version 1.4		05. may. 2012
programmer 		ks
tested by		ks

MB_SERVER ermöglicht das Lesen/Schreiben von Daten durch ein Remote-Device mittels Modbus over Ethernet (OpenModbus)

*)
(* read system time *)
tx := DWORD_TO_TIME(T_PLC_MS());

FOR i := 1 TO 10 DO
	IF VMAP[i].TIME_OUT > T#0s THEN
		VMAP[i].TIME_OUT := VMAP[i].TIME_OUT + tx - last_cycle;
	END_IF;
END_FOR;
last_cycle := tx;
ip_error := IP_C.ERROR > DWORD#0;

CASE state OF
00: (* Warten auf Freigabe *)
	IF ENABLE THEN
		state := 10;
		ip_state := BYTE#1; (* Anmelden *)
	END_IF;

10: (* Bei IP_Control anmelden und auf freigabe warten *)
	IF ip_state = BYTE#3 THEN

		(* IP Datenverkehr einrichten *)
		IP_C.C_PORT := WORD#0; (* Port von IP_CONTROL verwenden *)
		IP_C.C_IP := DWORD#0; (* IP von IP_CONTROL verwenden *)
		IP_C.C_MODE := SEL(UDP,BYTE#4,BYTE#5); (* Mode: 4=TCP+PASSIV+PORT , 5=UDP+PASSIV+PORT *)
		IP_C.TIME_RESET := TRUE; (* Zeitueberwachung rücksetzen *)
		IP_C.C_ENABLE := TRUE; (* Verbindungsaufbau freigeben *)
		IP_C.R_OBSERVE := TRUE; (* keine Empfangsueberwachung *)
		state := 20;
	END_IF;

20:	IF NOT ip_error THEN
		IF S_BUF.SIZE = UINT#0 AND R_BUF.SIZE > UINT#6 THEN	(* Datensenden nicht aktiv und Daten wurden empfangen *)
			IF  R_BUF.SIZE = WORD_TO_UINT(WORD_OF_BYTE(R_BUF.BUFFER[4],R_BUF.BUFFER[5])) + UINT#6 THEN (* gültige Datenlänge *)
				ERROR := DWORD#00; (* Error löschen *)

				(* Header kopieren *)
				FOR i := 0 TO 13 DO
					S_BUF.BUFFER[i] := R_BUF.BUFFER[i];
				END_FOR;
				fc := BYTE_TO_INT(R_BUF.BUFFER[7]);
				adr1 := WORD_TO_INT(WORD_OF_BYTE(R_BUF.BUFFER[8],R_BUF.BUFFER[9]));
				points := WORD_TO_INT(WORD_OF_BYTE(R_BUF.BUFFER[10],R_BUF.BUFFER[11]));

				(* Virtual Address *)
				MB_VMAP(VMAP:=VMAP,FC:=fc,V_ADR:=adr1,V_CNT:=points,SIZE:=DATA_SIZE);
				adr1:=MB_VMAP.P_ADR;
				bit_pos:=MB_VMAP.P_BIT;
				ERROR:=BYTE_TO_DWORD(MB_VMAP.ERROR);

				IF ERROR = DWORD#0 THEN
					CASE fc OF
					(*---------------------------------------------*)
					1..2 : (* Read Coil Status / Read Input Status *)
						count := 9; (* erstes Datenbyte *)
						coils := BYTE#0;
						mask := BYTE#1;
						FOR i := 1 TO points DO
							IF mask = BYTE#0 THEN
								mask := BYTE#1;
								S_BUF.BUFFER[count] := coils;
								coils := BYTE#0;
								count := count + 1;
							END_IF;
							IF (DATA[adr1] AND SHL(WORD#1,bit_pos)) > WORD#0 THEN
								coils := coils OR mask;
							END_IF;
	
							bit_Pos := bit_Pos + 1;
							IF bit_pos > 15 THEN
								ADR1 := ADR1 + 1;
								bit_pos := 0;
							END_IF;
	
							mask := SHL(mask,1);
						END_FOR;
						S_BUF.BUFFER[Count] := coils;
	
						S_BUF.BUFFER[8] := INT_TO_BYTE(count - 8); (* Bytecount *)
						S_BUF.SIZE := INT_TO_UINT(count + 1);
	
					(*--------------------------------------------------*)
					3..4 : (* Read Holding Registers / Read Input Registers *)
						idx1 := 07;
						count := adr1 + points - 1;
						FOR i := adr1 TO count DO
							idx1 := idx1 + 2;
							idx2 := idx1 + 1; (* zweiter index für pcworx notwendig ! *)
							w_tmp := DATA[i];
							S_BUF.BUFFER[idx1] := WORD_TO_BYTE(SHR(w_tmp,8));
							S_BUF.BUFFER[idx2] := WORD_TO_BYTE(w_tmp);
						END_FOR;
						S_BUF.BUFFER[8] := SHL(INT_TO_BYTE(points),1); (* Anzahl Register in Bytes *)
						S_BUF.SIZE := INT_TO_UINT(idx2 + 1);
					(*--------------------------------------------------*)
					5 : (* Force Single Coil *)
						DATA[adr1]:=BIT_LOAD_W(DATA[adr1],R_BUF.BUFFER[10] > BYTE#0,bit_pos);
						S_BUF.SIZE := UINT#12;
					(*--------------------------------------------------*)
					6 : (* Preset Single Register *)
						DATA[adr1] := WORD_OF_BYTE(R_BUF.BUFFER[10],R_BUF.BUFFER[11]);
						S_BUF.SIZE := UINT#12;
					(*--------------------------------------------------*)
					15 : (* Force Multible Coils *)
						mask := BYTE#1;
						idx1 := 13;
						FOR i := 1 TO points DO
							DATA[adr1]:=BIT_LOAD_W(DATA[adr1],(R_BUF.BUFFER[idx1] AND mask) > BYTE#0,bit_pos);
							bit_pos := bit_pos + 1;
							IF bit_pos > 15 THEN
								adr1:= adr1 + 1;
								bit_pos := 0;
							END_IF;
							mask := ROL(mask,1);
							IF mask = BYTE#1 THEN
								idx1 := idx1 +1;
							END_IF;
						END_FOR;
						S_BUF.SIZE := UINT#12;
					(*--------------------------------------------------*)
					16 : (* Preset Multiple Registers	*)
						idx1 := 11;
						count := adr1 + points - 1;
						FOR i := adr1 TO Count DO
							idx1 := idx1 + 2;
	 						idx2 := idx1 + 1;
							Data[i] := WORD_OF_BYTE(R_BUF.BUFFER[idx1],R_BUF.BUFFER[idx2]);
						END_FOR;
						S_BUF.SIZE := UINT#12;
					(*--------------------------------------------------*)
					22 : (* Mask Write Register *)
						w_tmp := WORD_OF_BYTE(R_BUF.BUFFER[10],R_BUF.BUFFER[11]); (* and mask *)
						DATA[adr1] := (DATA[adr1] AND w_tmp) OR (WORD_OF_BYTE(R_BUF.BUFFER[12],R_BUF.BUFFER[13]) AND (NOT w_tmp));
						S_BUF.SIZE := UINT#14;
					(*--------------------------------------------------*)
					23 : (* Read / Write Registers	*)
						(*--- Write-Register -----------------------------------*)
						adr2 := WORD_TO_INT(WORD_OF_BYTE(R_BUF.BUFFER[12],R_BUF.BUFFER[13]));
						points2 := WORD_TO_INT(WORD_OF_BYTE(R_BUF.BUFFER[14],R_BUF.BUFFER[15]));

						(* Virtual Address Write Register *)
						MB_VMAP(VMAP:=VMAP,FC:=16,V_ADR:=adr2,V_CNT:=points2,SIZE:=DATA_SIZE);
						adr2:=MB_VMAP.P_ADR;
						ERROR:=BYTE_TO_DWORD(MB_VMAP.ERROR);
	
						IF ERROR = DWORD#0 THEN
							idx1 := 15;
							count := adr2 + points2 - 1;
							FOR i := adr2 TO count DO
								idx1 := idx1 + 2;
	 							idx2 := idx1 + 1; (* zweiter index für pcworx notwendig ! *)
								Data[i] := WORD_OF_BYTE(R_BUF.BUFFER[idx1],R_BUF.BUFFER[idx2]);
							END_FOR;
	
							(*--- Read-Register -----------------------------------*)
							idx1 := 07;
							count := adr1 + points - 1;
							FOR i := adr1 TO count DO
								idx1 := idx1 + 2;
								idx2 := idx1 + 1; (* zweiter index für pcworx notwendig ! *)
								w_tmp := DATA[i];
								S_BUF.BUFFER[idx1] := WORD_TO_BYTE(SHR(w_tmp,8));
								S_BUF.BUFFER[idx2] := WORD_TO_BYTE(w_tmp);
							END_FOR;
							S_BUF.BUFFER[8] := SHL(INT_TO_BYTE(points),1); (* Anzahl Register in Bytes *)
							S_BUF.SIZE := INT_TO_UINT(idx2 + 1);
	
						END_IF;
	
					(*--------------------------------------------------*)
					ELSE
						ERROR := DWORD#01; (* ILLEGAL FUNCTION *)
					END_CASE;
				END_IF;
			END_IF;
	
			IF ERROR > DWORD#0 THEN
				S_BUF.BUFFER[7] := S_BUF.BUFFER[7] OR BYTE#2#1000_0000; (* Fehlerbit setzen *)
				S_BUF.BUFFER[8] := DWORD_TO_BYTE(ERROR);
				S_BUF.SIZE := UINT#9;
			END_IF;
	
			S_BUF.BUFFER[4] := BYTE#0; (* high Byte *)
			S_BUF.BUFFER[5] := UINT_TO_BYTE(S_BUF.SIZE - UINT#6); (* Längenfeld eintragen - nur low byte *)
	
		END_IF;
	ELSE
		ERROR := IP_C.ERROR;
	END_IF;

	t(IN:= ip_error, PT:=T#2s);
	IF t.Q THEN
		IP_C.TIME_RESET := TRUE; (* Error Reset *)
	END_IF;

	R_BUF.SIZE := UINT#0; (* Empfangsdaten zerstören *)

	IF ENABLE = FALSE OR t.Q THEN
	    ip_state := BYTE#4; (* Abmelden *)
		state := 00;
		IP_C.C_ENABLE := FALSE;
	END_IF;
END_CASE;

(* IP_FIFO *)
IP_FIFO(FIFO:=IP_C.FIFO,STATE:=ip_state,ID:=ip_id);

(* revision history
ks	05. jan. 2009	rev 1.0
	original version

ks	28. jan. 2009	rev 1.1
	network_buffer_short verwendet  

ks	20. oct. 2009	rev 1.2
	change lokal-var adr to adr1,Networkbuffer und Buffer-funktionen auf Basis 0

ks	17. may. 2011	rev 1.3
	automatischer re-connect

ks	05. may. 2012	rev 1.4
	timeoutüberwachung für re-connect
*)
END_FUNCTION_BLOCK

(* POU MD5_CRAM_AUTH_DEMO, CFC *)
PROGRAM MD5_CRAM_AUTH_DEMO
VAR
	run: BOOL := TRUE;
	timestamp : STRING(64) := 'PDQwMzYuMTA3NjMyNDM4MUBndWlsZGVuc3Rlcm4uemVpdGZvcm0uZGU+';
	password : STRING := 'geheimes_passwort';
	username : STRING := 'benutzer@zeitform.de';
	auth_key : STRING(STRING_LENGTH);
	MD5_CRAM_AUTH: MD5_CRAM_AUTH;
END_VAR
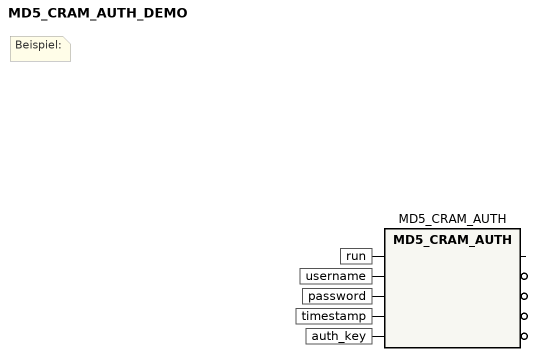
_CFC_ (* Continuous Function Chart, elements in execution order *)
#0 MD5_CRAM_AUTH:MD5_CRAM_AUTH(run, username, password, timestamp, auth_key)
(* Beispiel: *)
_END_CFC_
(* the same logic as Structured Text *)
MD5_CRAM_AUTH(run, username, password, timestamp, auth_key);
(* Beispiel: *)
END_PROGRAM

(* POU NET_VAR_MASTER_DEMO, CFC *)
PROGRAM NET_VAR_MASTER_DEMO
VAR
	NET_VAR_CONTROL_1: NET_VAR_CONTROL;
	activate: BOOL := TRUE;
	run: BOOL;
	udp: BOOL := TRUE;
	master: BOOL := TRUE;
	remote_port: WORD := 10000;
	scan_time: TIME := T#1s;
	watchdog: TIME := T#2s;
	error: DWORD;
	x: NET_VAR_DATA;

	NET_VAR_BOOL8_1: NET_VAR_BOOL8;
	id_b8: BYTE;
	in_b1: BOOL;
	in_b2: BOOL;
	in_b3: BOOL;
	in_b4: BOOL;
	in_b5: BOOL;
	in_b6: BOOL;
	in_b7: BOOL;
	in_b8: BOOL;
	out_b1: BOOL;
	out_b2: BOOL;
	out_b3: BOOL;
	out_b4: BOOL;
	out_b5: BOOL;
	out_b6: BOOL;
	out_b7: BOOL;
	out_b8: BOOL;

	NET_VAR_STRING_1: NET_VAR_STRING;
	in_s1: STRING(STRING_LENGTH);
	out_s1: STRING(STRING_LENGTH);
	id_s: BYTE;

	NET_VAR_BUFFER_1: NET_VAR_BUFFER;
	id_bu: BYTE;
	BUF_IN : ARRAY [1..64] OF BYTE;
	BUF_OUT : ARRAY [1..64] OF BYTE;

	id_dw: BYTE;
	NET_VAR_DWORD8_1: NET_VAR_DWORD8;
	in_dw1 : DWORD;
	in_dw2 : DWORD;
	in_dw3 : DWORD;
	in_dw4 : DWORD;
	in_dw5 : DWORD;
	in_dw6 : DWORD;
	in_dw7 : DWORD;
	in_dw8 : DWORD;
	out_dw1 : DWORD;
	out_dw2 : DWORD;
	out_dw3 : DWORD;
	out_dw4 : DWORD;
	out_dw5 : DWORD;
	out_dw6 : DWORD;
	out_dw7 : DWORD;
	out_dw8 : DWORD;

	NET_VAR_REAL8_1: NET_VAR_REAL8;
	in_r1 : REAL;
	in_r2 : REAL;
	in_r3 : REAL;
	in_r4 : REAL;
	in_r5 : REAL;
	in_r6 : REAL;
	in_r7 : REAL;
	in_r8 : REAL;
	out_r1 : REAL;
	out_r2 : REAL;
	out_r3 : REAL;
	out_r4 : REAL;
	out_r5 : REAL;
	out_r6 : REAL;
	out_r7 : REAL;
	out_r8 : REAL;
	id_r: BYTE;

	NET_VAR_X8_1: NET_VAR_X8;
	in_x_re1 : REAL;
	in_x_re2 : REAL;
	in_x_di1 : DINT;
	in_x_di2 : DINT;
	in_x_ud1 : UDINT;
	in_x_ud2 : UDINT;
	in_x_dw1 : DWORD;
	in_x_dw2 : DWORD;
	out_x_re1 : REAL;
	out_x_re2 : REAL;
	out_x_di1 : DINT;
	out_x_di2 : DINT;
	out_x_ud1 : UDINT;
	out_x_ud2 : UDINT;
	out_x_dw1 : DWORD;
	out_x_dw2 : DWORD;
	id_x8: BYTE;
END_VAR
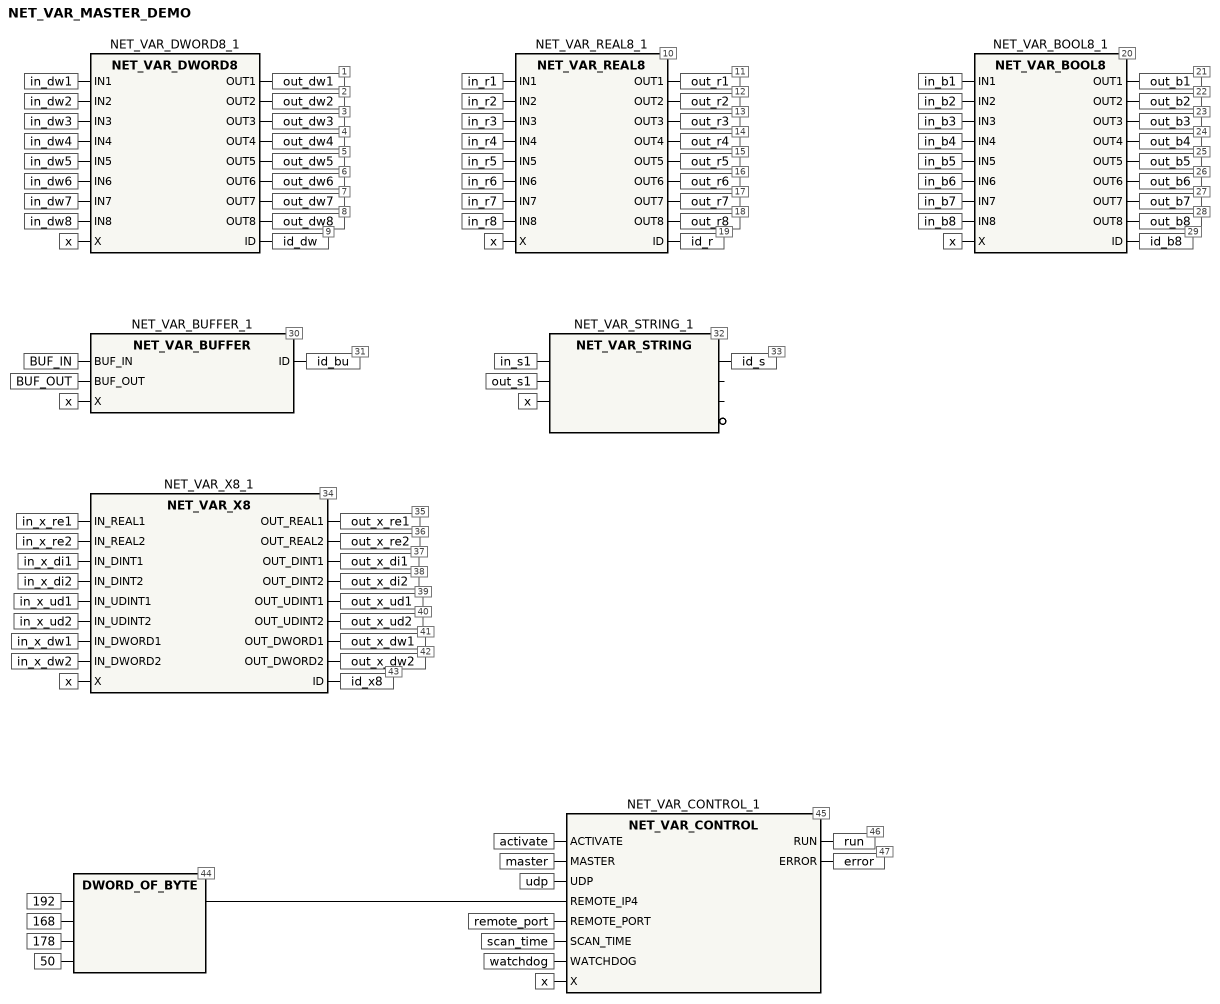
_CFC_ (* Continuous Function Chart, elements in execution order *)
#0 NET_VAR_DWORD8_1:NET_VAR_DWORD8(IN1: in_dw1, IN2: in_dw2, IN3: in_dw3, IN4: in_dw4, IN5: in_dw5, IN6: in_dw6, IN7: in_dw7, IN8: in_dw8, X: x)
#1 out_dw1 <= #0.OUT1
#2 out_dw2 <= #0.OUT2
#3 out_dw3 <= #0.OUT3
#4 out_dw4 <= #0.OUT4
#5 out_dw5 <= #0.OUT5
#6 out_dw6 <= #0.OUT6
#7 out_dw7 <= #0.OUT7
#8 out_dw8 <= #0.OUT8
#9 id_dw <= #0.ID
#10 NET_VAR_REAL8_1:NET_VAR_REAL8(IN1: in_r1, IN2: in_r2, IN3: in_r3, IN4: in_r4, IN5: in_r5, IN6: in_r6, IN7: in_r7, IN8: in_r8, X: x)
#11 out_r1 <= #10.OUT1
#12 out_r2 <= #10.OUT2
#13 out_r3 <= #10.OUT3
#14 out_r4 <= #10.OUT4
#15 out_r5 <= #10.OUT5
#16 out_r6 <= #10.OUT6
#17 out_r7 <= #10.OUT7
#18 out_r8 <= #10.OUT8
#19 id_r <= #10.ID
#20 NET_VAR_BOOL8_1:NET_VAR_BOOL8(IN1: in_b1, IN2: in_b2, IN3: in_b3, IN4: in_b4, IN5: in_b5, IN6: in_b6, IN7: in_b7, IN8: in_b8, X: x)
#21 out_b1 <= #20.OUT1
#22 out_b2 <= #20.OUT2
#23 out_b3 <= #20.OUT3
#24 out_b4 <= #20.OUT4
#25 out_b5 <= #20.OUT5
#26 out_b6 <= #20.OUT6
#27 out_b7 <= #20.OUT7
#28 out_b8 <= #20.OUT8
#29 id_b8 <= #20.ID
#30 NET_VAR_BUFFER_1:NET_VAR_BUFFER(BUF_IN: BUF_IN, BUF_OUT: BUF_OUT, X: x)
#31 id_bu <= #30.ID
#32 NET_VAR_STRING_1:NET_VAR_STRING(in_s1, out_s1, x)
#33 id_s <= #32.out 1
#34 NET_VAR_X8_1:NET_VAR_X8(IN_REAL1: in_x_re1, IN_REAL2: in_x_re2, IN_DINT1: in_x_di1, IN_DINT2: in_x_di2, IN_UDINT1: in_x_ud1, IN_UDINT2: in_x_ud2, IN_DWORD1: in_x_dw1, IN_DWORD2: in_x_dw2, X: x)
#35 out_x_re1 <= #34.OUT_REAL1
#36 out_x_re2 <= #34.OUT_REAL2
#37 out_x_di1 <= #34.OUT_DINT1
#38 out_x_di2 <= #34.OUT_DINT2
#39 out_x_ud1 <= #34.OUT_UDINT1
#40 out_x_ud2 <= #34.OUT_UDINT2
#41 out_x_dw1 <= #34.OUT_DWORD1
#42 out_x_dw2 <= #34.OUT_DWORD2
#43 id_x8 <= #34.ID
#44 DWORD_OF_BYTE(192, 168, 178, 50)
#45 NET_VAR_CONTROL_1:NET_VAR_CONTROL(ACTIVATE: activate, MASTER: master, UDP: udp, REMOTE_IP4: #44, REMOTE_PORT: remote_port, SCAN_TIME: scan_time, WATCHDOG: watchdog, X: x)
#46 run <= #45.RUN
#47 error <= #45.ERROR
_END_CFC_
END_PROGRAM

(* POU NET_VAR_CONTROL, ST *)
FUNCTION_BLOCK NET_VAR_CONTROL
VAR_INPUT
	ACTIVATE : BOOL;
	MASTER : BOOL;
	UDP : BOOL;
	REMOTE_IP4 : DWORD;
	REMOTE_PORT : WORD := 10000;
	SCAN_TIME : TIME := T#1s;
	WATCHDOG : TIME := T#2s;
END_VAR
VAR_OUTPUT
	RUN : BOOL;
	ERROR : DWORD;
END_VAR
VAR_IN_OUT
	X : NET_VAR_DATA;
END_VAR
VAR
	IPC : IP_CONTROL;
	IP_C : IP_C; (* IP_Control Verwaltungsstruktur *)
	step : INT;
	activate_last : BOOL;
	tscan : TON;
	reset : BOOL;
END_VAR

(*
version 1.0		15. may. 2011
programmer		ks
tested by			ks

NET_VAR_CONTROL überträgt Daten bidirektional vom Master zum Client
*)

(* Typ
001 = BYTE
002 = WORD
003 = DWORD
004 = BOOL (8x)
005 = REAL
006 = STRING
007 = UINT
008 = INT
009 = DINT
010 = UDINT
013 = DWORD (8x)
015 = REAL (8x)

020 = BUFFER
021 = MIX (REAL,DINT,UDINT,
*)
IF X.ERROR_ID > BYTE#0 THEN (* Schwere Fehler bei Variablenzuordnung vorhanden  !! *)
	X.STATE := BYTE#0;
	ERROR := BYTE_TO_DWORD(X.ERROR_ID);
	X.ERROR_ID := BYTE#0;
	step := 999;
END_IF;

CASE step OF

00:	IF ACTIVATE AND NOT activate_last OR reset THEN

        (*  TCP + MASTER = C_MODE 0 (TCP + ACTIVE + PORT + IP) *)
        (*  UDP + MASTER = C_MODE 1 (UDP + ACTIVE + PORT + IP) *)
        (*  TCP + SLAVE  = C_MODE 2 (TCP + PASSIV + PORT + IP) *)
        (*  UDP + SLAVE  = C_MODE 3 (UDP + PASSIV + PORT + IP) *)
	IF MASTER THEN
		IP_C.C_MODE := BYTE#0;
		step := 100;
	ELSE
		IP_C.C_MODE := BYTE#2;
		step := 200;
	END_IF;
        IF UDP THEN IP_C.C_MODE := IP_C.C_MODE OR BYTE#1; END_IF;
	  	IP_C.C_PORT := REMOTE_PORT; (* Portnummer eintragen *)
	  	IP_C.C_IP := REMOTE_IP4; (* IP eintragen *)
	  	IP_C.TIME_RESET := TRUE; (* Zeitueberwachung rücksetzen *)
	  	IP_C.C_ENABLE := TRUE; (* Verbindungsaufbau freigeben *)
	  	IP_C.R_OBSERVE := TRUE; (* Empfangsueberwachung *)
		X.S_BUF.SIZE := UINT#0;
		X.R_BUF.SIZE := UINT#0;
		X.CYCLE := UDINT#0;
		X.ERROR_ID := BYTE#0;
		reset := FALSE;
	END_IF;

(* ++++++++++++++++++++++++++++++++++++++++++++++ *)

100:IF IP_C.C_STATE > BYTE#127 THEN (* Verbindung vorhanden *)
		X.STATE := BYTE#1; (* Daten sammeln *)
		X.BUF_SIZE := SIZEOF(X.S_BUF.BUFFER);
		X.S_BUF.BUFFER[0] := UDINT_TO_BYTE(X.CYCLE);
		X.INDEX := 1;
		step := 110;
	END_IF;

110:X.STATE := BYTE#0;
	X.S_BUF.SIZE := INT_TO_UINT(X.INDEX); (* Datenlänge eintragen *)
	step := 120;

120:IF X.S_BUF.SIZE = UINT#0 AND X.R_BUF.SIZE >= UINT#1 THEN (* länge der empfangenen Daten prüfen *)
		X.STATE := BYTE#2; (* Daten ausgeben *)
		X.BUF_SIZE := X.R_BUF.SIZE;
		X.INDEX := 1;
		X.ERROR_ID := BYTE#0;
		X.CYCLE := X.CYCLE + UDINT#1;
		ERROR := DWORD#0; (* nach erfolgreichen Zyklus letzten Fehlercode löschen *)
		RUN := TRUE;
		step := 130;
	END_IF;

130:X.STATE := BYTE#0;
	X.R_BUF.SIZE := UINT#0;
	IF NOT ACTIVATE THEN
		step := 999; (* Beenden *)
	ELSIF tscan.Q THEN
		step := 100;
	END_IF;

(* ++++++++++++++++++++++++++++++++++++++++++++++ *)

200:IF X.R_BUF.SIZE >= UINT#1 THEN
		X.STATE := BYTE#2; (* Daten ausgeben *)
		X.BUF_SIZE := X.R_BUF.SIZE;
		X.INDEX := 1;
		step := 210;
	END_IF;

210:X.STATE := BYTE#1; (* Daten sammeln *)
	X.BUF_SIZE := SIZEOF(X.R_BUF.BUFFER);;
	X.S_BUF.BUFFER[0] := X.R_BUF.BUFFER[0]; (* Cycle übernehmen *)
	X.INDEX := 1;
	X.R_BUF.SIZE := UINT#0;
	step := 220;

220:X.STATE := BYTE#0;
	X.S_BUF.SIZE := INT_TO_UINT(X.INDEX); (* Datenlänge eintragen *)
	step := 230;

230:IF X.S_BUF.SIZE = UINT#0 THEN
		ERROR := DWORD#0; (* nach erfolgreichen Zyklus letzten Fehlercode löschen *)
		RUN := TRUE;
		IF NOT ACTIVATE THEN
			step := 999; (* Beenden *)
		ELSE
			step := 200;
		END_IF;
	END_IF;

999:IP_C.C_ENABLE := FALSE; (* Beenden *)
	RUN := FALSE;
	step := 0;

END_CASE;

(* ++++++++++++++++++++++++++++++++++++++++++++++ *)

IPC(IP:= DWORD#0, PORT:= WORD#0 , TIME_OUT:= WATCHDOG, IP_C:= IP_C, S_BUF:= X.S_BUF, R_BUF:= X.R_BUF);

IF IP_C.ERROR > DWORD#0 THEN
	ERROR := IP_C.ERROR;
	RUN := FALSE;
	reset := TRUE;
	step := 0;
END_IF;

ACTIVATE_LAST := ACTIVATE; (* letzten Status sichern zur Flankenerkennung *)
tscan(IN:= step <> 110 ,PT:=SCAN_TIME);

(* revision history
ks	15.may. 2011	rev 1.0
	original version

*)
END_FUNCTION_BLOCK

(* POU NET_VAR_BOOL8, ST *)
FUNCTION_BLOCK NET_VAR_BOOL8
VAR_IN_OUT
	X : NET_VAR_DATA;
END_VAR
VAR_INPUT
	IN1 : BOOL;
	IN2 : BOOL;
	IN3 : BOOL;
	IN4 : BOOL;
	IN5 : BOOL;
	IN6 : BOOL;
	IN7 : BOOL;
	IN8 : BOOL;
END_VAR
VAR_OUTPUT
	OUT1 : BOOL;
	OUT2 : BOOL;
	OUT3 : BOOL;
	OUT4 : BOOL;
	OUT5 : BOOL;
	OUT6 : BOOL;
	OUT7 : BOOL;
	OUT8 : BOOL;
	ID : BYTE;
END_VAR
VAR
	init : BOOL;
	index : INT;
	index2 : INT;
	BYTE_TO_BITS : BYTE_TO_BITS;
END_VAR

(*
version 1.0		15. may. 2011
programmer		ks
tested by			ks

NET_VAR_BOOL8 überträgt bidirektional 8 boolsche Werte vom Master zum Client
*)
IF NOT init THEN
	init := TRUE;
	X.ID_MAX := X.ID_MAX + USINT#1;
	ID := USINT_TO_BYTE(X.ID_MAX);
END_IF;

IF X.STATE > BYTE#0 AND X.ERROR_ID = BYTE#0 THEN
	index := X.index; (* PCWORX Workaround *)
	IF INT_TO_UINT(index + 3) > X.BUF_SIZE THEN
		X.ERROR_ID := ID;
	ELSE
		IF X.STATE = BYTE#1 THEN (* Daten schreiben *)
			X.S_BUF.BUFFER[index] := ID; (* ID *)
			index := index + 1;
			X.S_BUF.BUFFER[index] := BYTE#4; (* TYPE BOOL8 *)
			index := index + 1;
			X.S_BUF.BUFFER[index] := BYTE_OF_BIT(IN1,IN2,IN3,IN4,IN5,IN6,IN7,IN8);
			index := index + 1;

		ELSIF X.STATE = BYTE#2 THEN (* Daten lesen *)
			index2 := index + 1; (* PCWORX Workaround *)
			IF X.R_BUF.BUFFER[index] <> ID OR X.R_BUF.BUFFER[index2] <> BYTE#4 THEN
				X.ERROR_ID := ID;
			ELSE
				index := index + 2;
				BYTE_TO_BITS(IN:=X.R_BUF.BUFFER[index]);
				OUT1 := BYTE_TO_BITS.B0;
				OUT2 := BYTE_TO_BITS.B1;
				OUT3 := BYTE_TO_BITS.B2;
				OUT4 := BYTE_TO_BITS.B3;
				OUT5 := BYTE_TO_BITS.B4;
				OUT6 := BYTE_TO_BITS.B5;
				OUT7 := BYTE_TO_BITS.B6;
				OUT8 := BYTE_TO_BITS.B7;
				index := index + 1;
			END_IF;
		END_IF;
		X.index := index;
	END_IF;
END_IF;

(* revision history
ks	15.may. 2011	rev 1.0
	original version

*)
END_FUNCTION_BLOCK

(* POU NET_VAR_STRING, ST *)
FUNCTION_BLOCK NET_VAR_STRING
VAR_IN_OUT
	IN : STRING(STRING_LENGTH);
	OUT : STRING(STRING_LENGTH);
	X : NET_VAR_DATA;
END_VAR
VAR_OUTPUT
	ID : BYTE;
END_VAR
VAR
	init : BOOL;
	len_str : INT;
	index : INT;
	index2 : INT;
END_VAR

(*
version 1.0		15. may. 2011
programmer		ks
tested by			ks

NET_VAR_STRING überträgt bidirektional einen STRING vom Master zum Client
*)
IF NOT init THEN
	init := TRUE;
	X.ID_MAX := X.ID_MAX + USINT#1;
	ID := USINT_TO_BYTE(X.ID_MAX);
END_IF;

IF X.STATE > BYTE#0 AND X.ERROR_ID = BYTE#0 THEN
	index := X.index; (* PCWORX Workaround *)
	IF X.STATE = BYTE#1 THEN (* Daten schreiben *)
		len_str := LEN(IN);
		IF INT_TO_UINT(index + 3 + len_str) > X.BUF_SIZE THEN
			X.ERROR_ID := ID;
		ELSE
			X.S_BUF.BUFFER[index] := ID; (* ID *)
			index := index + 1;
			X.S_BUF.BUFFER[index] := BYTE#6; (* TYPE REAL *)
			index := index + 1;
			X.S_BUF.BUFFER[index] := INT_TO_BYTE(len_str); (* Anzahl der Bytes *)
			index := index + 1;
			_STRING_TO_BUFFER(STR:=IN,POS:=index,PT:=ADR(X.S_BUF.BUFFER),SIZE:=X.BUF_SIZE);
			index := index + len_str;
		END_IF;
	ELSIF X.STATE = BYTE#2 THEN (* Daten lesen *)
		index2 := index + 1; (* PCWORX Workaround *)
		IF X.R_BUF.BUFFER[index] <> ID OR X.R_BUF.BUFFER[index2] <> BYTE#6 THEN
			X.ERROR_ID := ID;
		ELSE
			index := index + 2;
			len_str := BYTE_TO_INT(X.R_BUF.BUFFER[index]);
			index2 := index + 1;
			index := index2 + len_str;
			IF len_STR > 0 THEN
				OUT := BUFFER_TO_STRING(PT:=ADR(X.R_BUF.BUFFER),SIZE:=X.BUF_SIZE,START:=INT_TO_UINT(index2),STOP:=INT_TO_UINT(index - 1));
			ELSE
				OUT := '';
			END_IF;
		END_IF;
	END_IF;
	X.index := index;
END_IF;

(* revision history
ks	15.may. 2011	rev 1.0
	original version

*)
END_FUNCTION_BLOCK

(* POU NET_VAR_BUFFER, ST *)
FUNCTION_BLOCK NET_VAR_BUFFER
VAR_IN_OUT
	BUF_IN : ARRAY[1..64] OF BYTE;
	BUF_OUT : ARRAY[1..64] OF BYTE;
	X : NET_VAR_DATA;
END_VAR
VAR_OUTPUT
	ID : BYTE;
END_VAR
VAR
	size : INT;
	init : BOOL;
	index : INT;
	index2 : INT;
END_VAR

(*
version 1.0		15. may. 2011
programmer		ks
tested by			ks

NET_VAR_BUFFER überträgt bidirektional 64 Bytes vom Master zum Client
*)
IF NOT init THEN
	init := TRUE;
	X.ID_MAX := X.ID_MAX + USINT#1;
	ID := USINT_TO_BYTE(X.ID_MAX);
END_IF;

IF X.STATE > BYTE#0 AND X.ERROR_ID = BYTE#0 THEN
	index := X.index; (* PCWORX Workaround *)
	IF X.STATE = BYTE#1 THEN (* Daten schreiben *)
		size := SIZEOF(BUF_IN);
		IF INT_TO_UINT(index + 3 + size) > X.BUF_SIZE THEN
			X.ERROR_ID := ID;
		ELSE
			X.S_BUF.BUFFER[index] := ID; (* ID *)
			index := index + 1;
			X.S_BUF.BUFFER[index] := BYTE#20; (* TYPE BUFFER *)
			index := index + 1;
			X.S_BUF.BUFFER[index] := INT_TO_BYTE(size); (* Anzahl der Bytes *)
				index := index + 1;
			FOR index2 := 1 TO size DO
				X.S_BUF.BUFFER[index] := BUF_IN[index2];
				index := index + 1;
			END_FOR;
		END_IF;
	ELSIF X.STATE = BYTE#2 THEN (* Daten lesen *)
		index2 := index + 1; (* PCWORX Workaround *)
		IF X.R_BUF.BUFFER[index] <> ID OR X.R_BUF.BUFFER[index2] <> BYTE#20 THEN
			X.ERROR_ID := ID;
		ELSE
			index := index + 2;
			size := BYTE_TO_INT(X.R_BUF.BUFFER[index]);
			index := index + 1;
			FOR index2 := 1 TO size DO
				BUF_OUT[index2] := X.R_BUF.BUFFER[index];
				index := index + 1;
			END_FOR;
		END_IF;
	END_IF;
	X.index := index;
END_IF;

(* revision history
ks	15.may. 2011	rev 1.0
	original version

*)
END_FUNCTION_BLOCK

(* POU NET_VAR_DWORD8, ST *)
FUNCTION_BLOCK NET_VAR_DWORD8
VAR_IN_OUT
	X : NET_VAR_DATA;
END_VAR
VAR_INPUT
	IN1 : DWORD;
	IN2 : DWORD;
	IN3 : DWORD;
	IN4 : DWORD;
	IN5 : DWORD;
	IN6 : DWORD;
	IN7 : DWORD;
	IN8 : DWORD;
END_VAR
VAR_OUTPUT
	OUT1 : DWORD;
	OUT2 : DWORD;
	OUT3 : DWORD;
	OUT4 : DWORD;
	OUT5 : DWORD;
	OUT6 : DWORD;
	OUT7 : DWORD;
	OUT8 : DWORD;
	ID : BYTE;
END_VAR
VAR
	init : BOOL;
	i : INT;
	i2 : INT;
	index : INT;
	index2 : INT;
	ra : ARRAY[1..8] OF DWORD;
END_VAR

(*
version 1.0		15. may. 2011
programmer		ks
tested by			ks

NET_VAR_DWORD8 überträgt bidirektional acht DWORD vom Master zum Client
*)
IF NOT init THEN
	init := TRUE;
	X.ID_MAX := X.ID_MAX + USINT#1;
	ID := USINT_TO_BYTE(X.ID_MAX);
END_IF;

IF X.STATE > BYTE#0 AND X.ERROR_ID = BYTE#0 THEN
	index := X.index; (* PCWORX Workaround *)
	IF INT_TO_UINT(index + 34) > X.BUF_SIZE THEN  (* ID (1) + TYPE (1) + 8 x DWORD (4) *)
		X.ERROR_ID := ID;
	ELSE
		IF X.STATE = BYTE#1 THEN (* Daten schreiben *)
			ra[1] := IN1;
			ra[2] := IN2;
			ra[3] := IN3;
			ra[4] := IN4;
			ra[5] := IN5;
			ra[6] := IN6;
			ra[7] := IN7;
			ra[8] := IN8;
			X.S_BUF.BUFFER[index] := ID; (* ID *)
			index := index + 1;
			X.S_BUF.BUFFER[index] := BYTE#13; (* TYPE DWORD8 *)
			index := index + 1;
			FOR i2 := 1 TO 8 DO;
				FOR i := 1 TO 4 DO;
					X.S_BUF.BUFFER[index] := DWORD_TO_BYTE(ra[i2]);
					ra[i2] := ROR(ra[i2],8);
					index := index + 1;
				END_FOR;
			END_FOR;

		ELSIF X.STATE = BYTE#2 THEN (* Daten lesen *)
			index2 := index + 1; (* PCWORX Workaround *)
			IF X.R_BUF.BUFFER[index] <> ID OR X.R_BUF.BUFFER[index2] <> BYTE#13 THEN (* TYPE DWORD8 *)
				X.ERROR_ID := ID;
			ELSE
				index := index + 2;
				FOR i2 := 1 TO 8 DO;
					ra[i2] := DWORD#0;
					FOR i := 1 TO 4 DO;
						ra[i2] := ra[i2] OR BYTE_TO_DWORD(X.R_BUF.BUFFER[index]);
						ra[i2] := ROR(ra[i2],8);
						index := index + 1;
					END_FOR;
				END_FOR;
				OUT1 := ra[1];
				OUT2 := ra[2];
				OUT3 := ra[3];
				OUT4 := ra[4];
				OUT5 := ra[5];
				OUT6 := ra[6];
				OUT7 := ra[7];
				OUT8 := ra[8];
			END_IF;
		END_IF;
		X.index := index;
	END_IF;
END_IF;

(* revision history
ks	15.may. 2011	rev 1.0
	original version

*)
END_FUNCTION_BLOCK

(* POU NET_VAR_REAL8, ST *)
FUNCTION_BLOCK NET_VAR_REAL8
VAR_IN_OUT
	X : NET_VAR_DATA;
END_VAR
VAR_INPUT
	IN1 : REAL;
	IN2 : REAL;
	IN3 : REAL;
	IN4 : REAL;
	IN5 : REAL;
	IN6 : REAL;
	IN7 : REAL;
	IN8 : REAL;
END_VAR
VAR_OUTPUT
	OUT1 : REAL;
	OUT2 : REAL;
	OUT3 : REAL;
	OUT4 : REAL;
	OUT5 : REAL;
	OUT6 : REAL;
	OUT7 : REAL;
	OUT8 : REAL;
	ID : BYTE;
END_VAR
VAR
	init : BOOL;
	i : INT;
	i2 : INT;
	index : INT;
	index2 : INT;
	r_dw : DWORD;
	ra : ARRAY[1..8] OF REAL;
END_VAR

(*
version 1.0		15. may. 2011
programmer		ks
tested by			ks

NET_VAR_REAL8 überträgt bidirektional acht REAL-Werte vom Master zum Client
*)
IF NOT init THEN
	init := TRUE;
	X.ID_MAX := X.ID_MAX + USINT#1;
	ID := USINT_TO_BYTE(X.ID_MAX);
END_IF;

IF X.STATE > BYTE#0 AND X.ERROR_ID = BYTE#0 THEN
	index := X.index; (* PCWORX Workaround *)
	IF INT_TO_UINT(index + 34) > X.BUF_SIZE THEN (* ID (1) + TYPE (1) + 8 x REAL (4) *)
		X.ERROR_ID := ID;
	ELSE
		IF X.STATE = BYTE#1 THEN (* Daten schreiben *)
			ra[1] := IN1;
			ra[2] := IN2;
			ra[3] := IN3;
			ra[4] := IN4;
			ra[5] := IN5;
			ra[6] := IN6;
			ra[7] := IN7;
			ra[8] := IN8;
			X.S_BUF.BUFFER[index] := ID; (* ID *)
			index := index + 1;
			X.S_BUF.BUFFER[index] := BYTE#15; (* TYPE REAL8 *)
			index := index + 1;
			FOR i2 := 1 TO 8 DO;
				r_dw := REAL_TO_DW(X:=ra[i2]);
				FOR i := 1 TO 4 DO;
					X.S_BUF.BUFFER[index] := DWORD_TO_BYTE(r_dw);
					r_dw := ROR(r_dw,8);
					index := index + 1;
				END_FOR;
			END_FOR;

		ELSIF X.STATE = BYTE#2 THEN (* Daten lesen *)
			index2 := index + 1; (* PCWORX Workaround *)
			IF X.R_BUF.BUFFER[index] <> ID OR X.R_BUF.BUFFER[index2] <> BYTE#15 THEN (* TYPE REAL8 *)
				X.ERROR_ID := ID;
			ELSE
				index := index + 2;
				FOR i2 := 1 TO 8 DO;
					r_dw := DWORD#0;
					FOR i := 1 TO 4 DO;
						r_dw := r_dw OR BYTE_TO_DWORD(X.R_BUF.BUFFER[index]);
						r_dw := ROR(r_dw,8);
						index := index + 1;
					END_FOR;
					ra[i2] := DW_TO_REAL(X:=r_dw);
				END_FOR;
				OUT1 := ra[1];
				OUT2 := ra[2];
				OUT3 := ra[3];
				OUT4 := ra[4];
				OUT5 := ra[5];
				OUT6 := ra[6];
				OUT7 := ra[7];
				OUT8 := ra[8];
			END_IF;
		END_IF;
		X.index := index;
	END_IF;
END_IF;

(* revision history
ks	15.may. 2011	rev 1.0
	original version

*)
END_FUNCTION_BLOCK

(* POU NET_VAR_X8, ST *)
FUNCTION_BLOCK NET_VAR_X8
VAR_IN_OUT
	X : NET_VAR_DATA;
END_VAR
VAR_INPUT
	IN_REAL1 : REAL;
	IN_REAL2 : REAL;
	IN_DINT1 : DINT;
	IN_DINT2 : DINT;
	IN_UDINT1 : UDINT;
	IN_UDINT2 : UDINT;
	IN_DWORD1 : DWORD;
	IN_DWORD2 : DWORD;
END_VAR
VAR_OUTPUT
	OUT_REAL1 : REAL;
	OUT_REAL2: REAL;
	OUT_DINT1 : DINT;
	OUT_DINT2 : DINT;
	OUT_UDINT1 : UDINT;
	OUT_UDINT2 : UDINT;
	OUT_DWORD1 : DWORD;
	OUT_DWORD2 : DWORD;
	ID : BYTE;
END_VAR
VAR
	init : BOOL;
	i : INT;
	i2 : INT;
	index : INT;
	index2 : INT;
	ra : ARRAY[1..8] OF DWORD;
END_VAR

(*
version 1.0		15. may. 2011
programmer		ks
tested by			ks

NET_VAR_X8 überträgt bidirektional 2x REAL,2x DINT,2x UDINT,2x DWORD vom Master zum Client
*)
IF NOT init THEN
	init := TRUE;
	X.ID_MAX := X.ID_MAX + USINT#1;
	ID := USINT_TO_BYTE(X.ID_MAX);
END_IF;

IF X.STATE > BYTE#0 AND X.ERROR_ID = BYTE#0 THEN
	index := X.index; (* PCWORX Workaround *)
	IF INT_TO_UINT(index + 34) > X.BUF_SIZE THEN  (* ID (1) + TYPE (1) + 8 x DWORD (4) *)
		X.ERROR_ID := ID;
	ELSE
		IF X.STATE = BYTE#1 THEN (* Daten schreiben *)
			ra[1] := REAL_TO_DW(X:=IN_REAL1);
			ra[2] := REAL_TO_DW(X:=IN_REAL2);
			ra[3] := DINT_TO_DWORD(IN_DINT1);
			ra[4] := DINT_TO_DWORD(IN_DINT2);
			ra[5] := UDINT_TO_DWORD(IN_UDINT1);
			ra[6] := UDINT_TO_DWORD(IN_UDINT2);
			ra[7] := IN_DWORD1;
			ra[8] := IN_DWORD2;
			X.S_BUF.BUFFER[index] := ID; (* ID *)
			index := index + 1;
			X.S_BUF.BUFFER[index] := BYTE#21; (* TYPE X8 *)
			index := index + 1;
			FOR i2 := 1 TO 8 DO;
				FOR i := 1 TO 4 DO;
					X.S_BUF.BUFFER[index] := DWORD_TO_BYTE(ra[i2]);
					ra[i2] := ROR(ra[i2],8);
					index := index + 1;
				END_FOR;
			END_FOR;

		ELSIF X.STATE = BYTE#2 THEN (* Daten lesen *)
			index2 := index + 1; (* PCWORX Workaround *)
			IF X.R_BUF.BUFFER[index] <> ID OR X.R_BUF.BUFFER[index2] <> BYTE#21 THEN (* TYPE X8 *)
				X.ERROR_ID := ID;
			ELSE
				index := index + 2;
				FOR i2 := 1 TO 8 DO;
					ra[i2] := DWORD#0;
					FOR i := 1 TO 4 DO;
						ra[i2] := ra[i2] OR BYTE_TO_DWORD(X.R_BUF.BUFFER[index]);
						ra[i2] := ROR(ra[i2],8);
						index := index + 1;
					END_FOR;
				END_FOR;
				OUT_REAL1 := DW_TO_REAL(X:=ra[1]);
				OUT_REAL2 := DW_TO_REAL(X:=ra[2]);
				OUT_DINT1 := DWORD_TO_DINT(ra[3]);
				OUT_DINT2 := DWORD_TO_DINT(ra[4]);
				OUT_UDINT1 := DWORD_TO_UDINT(ra[5]);
				OUT_UDINT2 := DWORD_TO_UDINT(ra[6]);
				OUT_DWORD1 := ra[7];
				OUT_DWORD2 := ra[8];
			END_IF;
		END_IF;
		X.index := index;
	END_IF;
END_IF;

(* revision history
ks	15.may. 2011	rev 1.0
	original version

*)
END_FUNCTION_BLOCK

(* POU NET_VAR_SLAVE_DEMO, CFC *)
PROGRAM NET_VAR_SLAVE_DEMO
VAR
	NET_VAR_CONTROL_1: NET_VAR_CONTROL;
	activate: BOOL := TRUE;
	run: BOOL;
	udp: BOOL := TRUE;
	master: BOOL := FALSE;
	remote_port: WORD := 10000;
	scan_time: TIME := T#1s;
	watchdog: TIME := T#2s;
	error: DWORD;
	x: NET_VAR_DATA;

	NET_VAR_BOOL8_1: NET_VAR_BOOL8;
	id_b8: BYTE;
	in_b1: BOOL;
	in_b2: BOOL;
	in_b3: BOOL;
	in_b4: BOOL;
	in_b5: BOOL;
	in_b6: BOOL;
	in_b7: BOOL;
	in_b8: BOOL;
	out_b1: BOOL;
	out_b2: BOOL;
	out_b3: BOOL;
	out_b4: BOOL;
	out_b5: BOOL;
	out_b6: BOOL;
	out_b7: BOOL;
	out_b8: BOOL;

	NET_VAR_STRING_1: NET_VAR_STRING;
	in_s1: STRING(STRING_LENGTH);
	out_s1: STRING(STRING_LENGTH);
	id_s: BYTE;

	NET_VAR_BUFFER_1: NET_VAR_BUFFER;
	id_bu: BYTE;
	BUF_IN : ARRAY [1..64] OF BYTE;
	BUF_OUT : ARRAY [1..64] OF BYTE;

	id_dw: BYTE;
	NET_VAR_DWORD8_1: NET_VAR_DWORD8;
	in_dw1 : DWORD;
	in_dw2 : DWORD;
	in_dw3 : DWORD;
	in_dw4 : DWORD;
	in_dw5 : DWORD;
	in_dw6 : DWORD;
	in_dw7 : DWORD;
	in_dw8 : DWORD;
	out_dw1 : DWORD;
	out_dw2 : DWORD;
	out_dw3 : DWORD;
	out_dw4 : DWORD;
	out_dw5 : DWORD;
	out_dw6 : DWORD;
	out_dw7 : DWORD;
	out_dw8 : DWORD;

	NET_VAR_REAL8_1: NET_VAR_REAL8;
	in_r1 : REAL;
	in_r2 : REAL;
	in_r3 : REAL;
	in_r4 : REAL;
	in_r5 : REAL;
	in_r6 : REAL;
	in_r7 : REAL;
	in_r8 : REAL;
	out_r1 : REAL;
	out_r2 : REAL;
	out_r3 : REAL;
	out_r4 : REAL;
	out_r5 : REAL;
	out_r6 : REAL;
	out_r7 : REAL;
	out_r8 : REAL;
	id_r: BYTE;

	NET_VAR_X8_1: NET_VAR_X8;
	in_x_re1 : REAL;
	in_x_re2 : REAL;
	in_x_di1 : DINT;
	in_x_di2 : DINT;
	in_x_ud1 : UDINT;
	in_x_ud2 : UDINT;
	in_x_dw1 : DWORD;
	in_x_dw2 : DWORD;
	out_x_re1 : REAL;
	out_x_re2 : REAL;
	out_x_di1 : DINT;
	out_x_di2 : DINT;
	out_x_ud1 : UDINT;
	out_x_ud2 : UDINT;
	out_x_dw1 : DWORD;
	out_x_dw2 : DWORD;
	id_x8: BYTE;
END_VAR
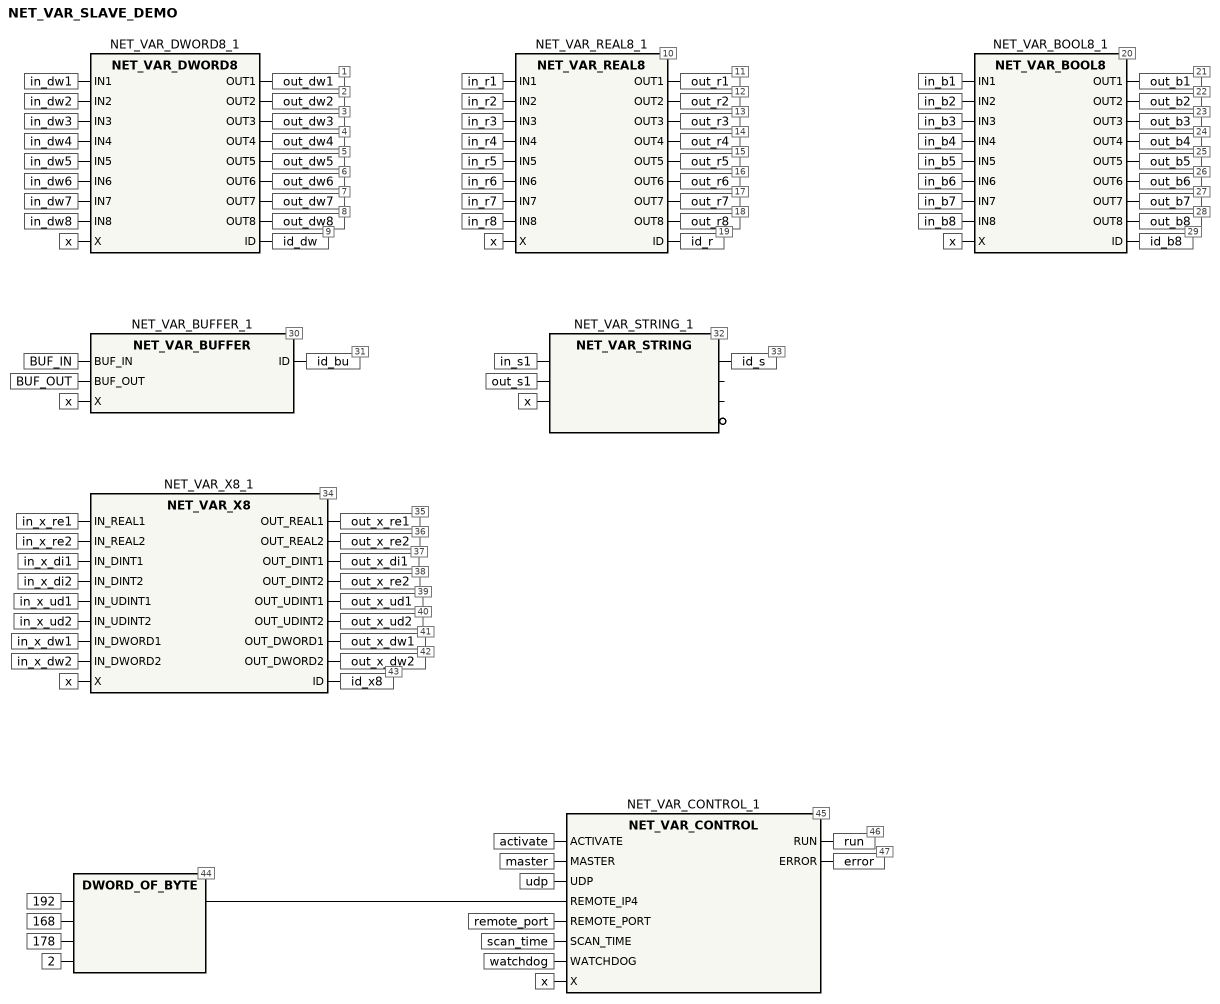
_CFC_ (* Continuous Function Chart, elements in execution order *)
#0 NET_VAR_DWORD8_1:NET_VAR_DWORD8(IN1: in_dw1, IN2: in_dw2, IN3: in_dw3, IN4: in_dw4, IN5: in_dw5, IN6: in_dw6, IN7: in_dw7, IN8: in_dw8, X: x)
#1 out_dw1 <= #0.OUT1
#2 out_dw2 <= #0.OUT2
#3 out_dw3 <= #0.OUT3
#4 out_dw4 <= #0.OUT4
#5 out_dw5 <= #0.OUT5
#6 out_dw6 <= #0.OUT6
#7 out_dw7 <= #0.OUT7
#8 out_dw8 <= #0.OUT8
#9 id_dw <= #0.ID
#10 NET_VAR_REAL8_1:NET_VAR_REAL8(IN1: in_r1, IN2: in_r2, IN3: in_r3, IN4: in_r4, IN5: in_r5, IN6: in_r6, IN7: in_r7, IN8: in_r8, X: x)
#11 out_r1 <= #10.OUT1
#12 out_r2 <= #10.OUT2
#13 out_r3 <= #10.OUT3
#14 out_r4 <= #10.OUT4
#15 out_r5 <= #10.OUT5
#16 out_r6 <= #10.OUT6
#17 out_r7 <= #10.OUT7
#18 out_r8 <= #10.OUT8
#19 id_r <= #10.ID
#20 NET_VAR_BOOL8_1:NET_VAR_BOOL8(IN1: in_b1, IN2: in_b2, IN3: in_b3, IN4: in_b4, IN5: in_b5, IN6: in_b6, IN7: in_b7, IN8: in_b8, X: x)
#21 out_b1 <= #20.OUT1
#22 out_b2 <= #20.OUT2
#23 out_b3 <= #20.OUT3
#24 out_b4 <= #20.OUT4
#25 out_b5 <= #20.OUT5
#26 out_b6 <= #20.OUT6
#27 out_b7 <= #20.OUT7
#28 out_b8 <= #20.OUT8
#29 id_b8 <= #20.ID
#30 NET_VAR_BUFFER_1:NET_VAR_BUFFER(BUF_IN: BUF_IN, BUF_OUT: BUF_OUT, X: x)
#31 id_bu <= #30.ID
#32 NET_VAR_STRING_1:NET_VAR_STRING(in_s1, out_s1, x)
#33 id_s <= #32.out 1
#34 NET_VAR_X8_1:NET_VAR_X8(IN_REAL1: in_x_re1, IN_REAL2: in_x_re2, IN_DINT1: in_x_di1, IN_DINT2: in_x_di2, IN_UDINT1: in_x_ud1, IN_UDINT2: in_x_ud2, IN_DWORD1: in_x_dw1, IN_DWORD2: in_x_dw2, X: x)
#35 out_x_re1 <= #34.OUT_REAL1
#36 out_x_re2 <= #34.OUT_REAL2
#37 out_x_di1 <= #34.OUT_DINT1
#38 out_x_re2 <= #34.OUT_DINT2
#39 out_x_ud1 <= #34.OUT_UDINT1
#40 out_x_ud2 <= #34.OUT_UDINT2
#41 out_x_dw1 <= #34.OUT_DWORD1
#42 out_x_dw2 <= #34.OUT_DWORD2
#43 id_x8 <= #34.ID
#44 DWORD_OF_BYTE(192, 168, 178, 2)
#45 NET_VAR_CONTROL_1:NET_VAR_CONTROL(ACTIVATE: activate, MASTER: master, UDP: udp, REMOTE_IP4: #44, REMOTE_PORT: remote_port, SCAN_TIME: scan_time, WATCHDOG: watchdog, X: x)
#46 run <= #45.RUN
#47 error <= #45.ERROR
_END_CFC_
END_PROGRAM

(* POU RC4_CRYPT_DEMO, CFC *)
PROGRAM RC4_CRYPT_DEMO
VAR
	RC4_CRYPT_STREAM: RC4_CRYPT_STREAM;
	(* buf : ARRAY [0..63] OF BYTE := 107,117,114,116;*) (* kurt *)
	buf : ARRAY [0..63] OF BYTE := 110,60,3,219; (* crypt *)
	mode: INT;
	key: STRING := '1234';
	size: UDINT := 4;
	pos: UDINT;
END_VAR
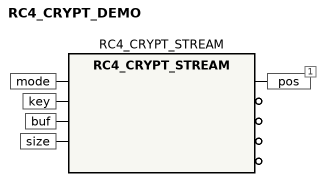
_CFC_ (* Continuous Function Chart, elements in execution order *)
#0 RC4_CRYPT_STREAM:RC4_CRYPT_STREAM(mode, key, buf, size)
#1 pos <= #0.out 1
_END_CFC_
END_PROGRAM

(* POU RC4_CRYPT_STREAM, ST *)
FUNCTION_BLOCK RC4_CRYPT_STREAM
VAR_IN_OUT
	MODE : INT;
	KEY : STRING(40);
	BUF : ARRAY [0..63] OF BYTE;
	SIZE : UDINT;
END_VAR

VAR_OUTPUT
	POS : UDINT;
END_VAR

VAR
	sbox : ARRAY [0..255] OF BYTE;
	skey : ARRAY [0..255] OF BYTE;
	a : INT;
	b : INT;
	c : INT;
	d : USINT;
	e : USINT;
	end : UDINT;
	v : BYTE;
END_VAR

(*
version 1.0	09. jan. 2010
programmer	ks
tested BY	ks

RC4_CRYPT_STREAM kann einen Datenstrom ver/entschlüsseln mittels der RC4 Stromchiffrierung
*)
CASE MODE OF

1:	(* Initialisierung *)
	b := LEN(KEY) - 1;
	IF b < 0 OR SIZE < 1 THEN
		MODE := 3;
		RETURN;
	END_IF;

	FOR a := 0 TO b DO
		skey[a] := CODE(KEY, a + 1);
		sbox[a] := INT_TO_BYTE(a);
	END_FOR;

	c := 0;
	FOR a := b + 1 TO 255 DO
		skey[a] := skey[c];
		sbox[a] := INT_TO_BYTE(a);
		c := c + 1;
		IF c > b THEN c := 0; END_IF;
	END_FOR;

	d := 0;
	FOR a := 0 TO 255 DO
		d := d + sbox[a] + skey[a];
		v := sbox[a];
		sbox[a] := sbox[d];
		sbox[d] := v;
	END_FOR;

	POS := 0;
	end := SIZE;
	SIZE := MIN(64,end);
	d := 0;
	e := 0;
	MODE := 2;

2:	(* Daten ver/entschlüsseln *)

	b := UDINT_TO_INT(SIZE) - 1;
	FOR a := 0 TO b DO
		d := d + 1;
		e := e + sbox[d];
		v := sbox[d];
		sbox[d] := sbox[e];
		sbox[e] := v;
		v := sbox[d] + sbox[e];
		BUF[a] :=BUF[a] XOR sbox[v];
	END_FOR;

	POS := POS + SIZE;
	SIZE := MIN(64,end - POS);

	IF SIZE = 0 THEN
		MODE := 3;
	END_IF;
END_CASE;

(* revision history

ks	9. Jan. 2010 rev 1.0
	original version

*)
END_FUNCTION_BLOCK

(* POU SHA1_MD5_DEMO, CFC *)
PROGRAM SHA1_MD5_DEMO
VAR
	text: STRING(STRING_LENGTH) := '<4036.1076324381@guildenstern.zeitform.de>';
	MD5_STR : MD5_STR;
	SHA1_STR : SHA1_STR;
	md5_hash : ARRAY [0..15] OF BYTE;
	sha1_hash : ARRAY [0..19] OF BYTE;
	start1 : BOOL := TRUE;
	start2 : BOOL := TRUE;
	done1 : BOOL;
	done2 : BOOL;
	md5_strh : STRING(32);
	sha1_strh : STRING(40);
END_VAR
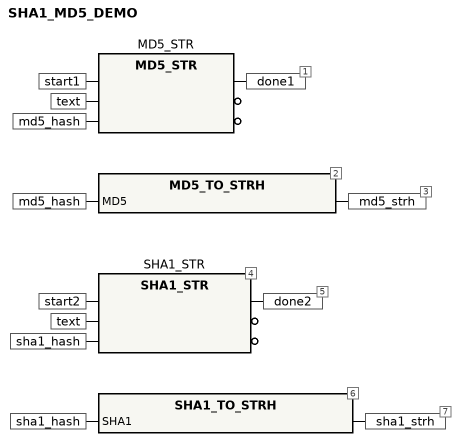
_CFC_ (* Continuous Function Chart, elements in execution order *)
#0 MD5_STR:MD5_STR(start1, text, md5_hash)
#1 done1 <= #0.out 1
#2 MD5_TO_STRH(MD5: md5_hash)
#3 md5_strh <= #2
#4 SHA1_STR:SHA1_STR(start2, text, sha1_hash)
#5 done2 <= #4.out 1
#6 SHA1_TO_STRH(SHA1: sha1_hash)
#7 sha1_strh <= #6
_END_CFC_
END_PROGRAM

(* POU MD5_STR, ST *)
FUNCTION_BLOCK MD5_STR
VAR_INPUT
	RUN: BOOL;
END_VAR
VAR_OUTPUT
	DONE: BOOL;
END_VAR
VAR_IN_OUT
	STR: STRING(STRING_LENGTH);
	MD5 : ARRAY [0..15] OF BYTE;
END_VAR
VAR
	run_last: BOOL;
	MD5_STREAM : MD5_STREAM;
	buf : ARRAY [0..63] OF BYTE;
	mode : INT;
	size : UDINT;
	pos : UDINT;
END_VAR

(*
version 1.0	06. dec. 2009
programmer 	ks
tested BY	ks

MD5_STR berechnet den MD5 Hash eines Strings
*)
CASE mode OF
0:	(* Wait für Start *)
	IF RUN AND NOT run_last THEN
		DONE := FALSE;
		mode := 1; (* Initialisierung *)
		size := LEN(STR);
	END_IF;

2:	(* Data copy and Calc *)
	IF size > 0 THEN
		_STRING_TO_BUFFER(STR:=MID(STR, UDINT_TO_INT(SIZE), UDINT_TO_INT(POS) + 1), POS:=0, PT:=ADR(buf), SIZE:=SIZEOF(buf));
	END_IF;

3:	DONE := TRUE;
	mode := 0; (* Stop *)

END_CASE;

IF mode > 0 THEN
	MD5_STREAM(SIZE:=size, MODE:=mode, BUF:=buf, MD5:=MD5, POS=>pos);
END_IF;

run_last := RUN;

(* revision history

ks	6. dec. 2009 rev 1.0
	original version

*)
END_FUNCTION_BLOCK

(* POU SHA1_STR, ST *)
FUNCTION_BLOCK SHA1_STR
VAR_INPUT
	RUN: BOOL;
END_VAR
VAR_OUTPUT
	DONE: BOOL;
END_VAR
VAR_IN_OUT
	STR: STRING(STRING_LENGTH);
	SHA1 : ARRAY [0..19] OF BYTE;
END_VAR

VAR
	run_last: BOOL;
	SHA1_STREAM : SHA1_STREAM;
	buf : ARRAY [0..63] OF BYTE;
	mode : INT;
	size : UDINT;
	pos : UDINT;
END_VAR

(*
version 1.0	06. dec. 2009
programmer 	ks
tested BY	ks

SHA1_STR berechnet den MD5 Hash eines Strings
*)
CASE mode OF
0:	(* Wait für Start *)
	IF RUN AND NOT run_last THEN
		DONE := FALSE;
		mode := 1; (* Initialisierung *)
		size := LEN(STR);
	END_IF;

2:	(* Data copy and Calc *)
	IF size > 0 THEN
		_STRING_TO_BUFFER(STR:=MID(STR, UDINT_TO_INT(SIZE), UDINT_TO_INT(POS) + 1), POS:=0, PT:=ADR(buf), SIZE:=SIZEOF(buf));
	END_IF;

3:	DONE := TRUE;
	mode := 0; (* Stop *)

END_CASE;

IF mode > 0 THEN
	SHA1_STREAM(SIZE:=size, MODE:=mode, BUF:=buf, SHA1:=SHA1, POS=>pos);
END_IF;

run_last := RUN;

(* revision history

ks	6. dec. 2009 rev 1.0
	original version

*)
END_FUNCTION_BLOCK

(* POU SHA1_TO_STRH, ST *)
FUNCTION SHA1_TO_STRH : STRING(40)
VAR_INPUT
	SHA1 : ARRAY [0..19] OF BYTE;
END_VAR
VAR
	i : INT;
	tmp : BYTE;
	pt : POINTER TO BYTE;
END_VAR
(*
version 1.1	03. dec. 2011
programmer 	ks
tested BY	ks

SHA1_TO_STRH konvertiert das SHA1 Hash Array in einen HEX-String
*)
pt := ADR(SHA1_TO_STRH); (* read output adress to pointer *)

FOR i := 0 TO 19 DO; (* write the 10 hex characters backwards *)
	tmp := SHR(SHA1[i],4);
	PT^ := tmp + SEL(tmp <= 9,87,48);
	pt := pt + 1; (* decrement the pointer *)
	tmp := SHA1[i] AND 2#1111;
	PT^ := tmp + SEL(tmp <= 9,87,48);
	pt := pt + 1; (* decrement the pointer *)
END_FOR;
pt^:= 0; (* write the closing byte for the string *)

(* revision history

ks	6. dec. 2009 rev 1.0
	original version

ks	3. dec. 2011 rev 1.1
	incorrect string size
*)
END_FUNCTION

(* POU SMTP_CLIENT_DEMO, CFC *)
PROGRAM SMTP_CLIENT_DEMO
VAR
(*
	smtp_server: STRING := 'oscat_test%freenet.de:oscat123456@mx.freenet.de';
	smtp_mailfrom: STRING := 'oscat_test@freenet.de';
*)

	SMTP_CLIENT: SMTP_CLIENT;
	smtp_activate: BOOL;
	smtp_timeout: TIME := T#30s;
	smtp_error_t: BYTE;
	smtp_error_c: DWORD;
	smtp_busy: BOOL;
	smtp_done: BOOL;
	smtp_dti: DT;
	smtp_dti_offset: INT := 60;
	smtp_files: STRING(STRING_LENGTH) := '';
	smtp_server: STRING := '110876022:oscat123456@mail.gmx.net';
	smtp_mailfrom: STRING := 'oscat@gmx.net;Station_01';
	smtp_mailto: STRING(STRING_LENGTH) := 'oscat@gmx.net';
	smtp_subject: STRING := 'Das ist der Betreff';
	smtp_body: STRING(STRING_LENGTH) := 'Das ist der Email-Text';
END_VAR
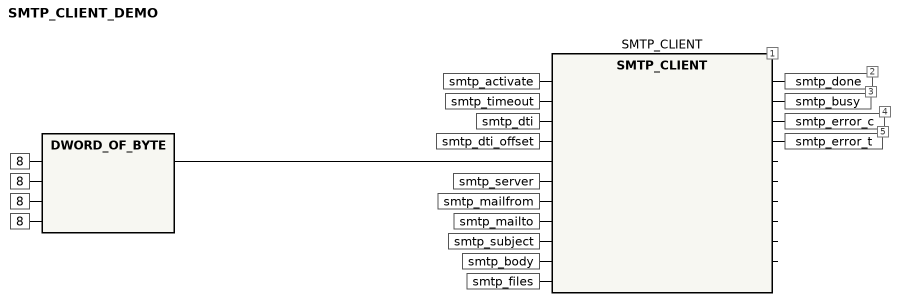
_CFC_ (* Continuous Function Chart, elements in execution order *)
#0 DWORD_OF_BYTE(8, 8, 8, 8)
#1 SMTP_CLIENT:SMTP_CLIENT(smtp_activate, smtp_timeout, smtp_dti, smtp_dti_offset, #0, smtp_server, smtp_mailfrom, smtp_mailto, smtp_subject, smtp_body, smtp_files)
#2 smtp_done <= #1.out 1
#3 smtp_busy <= #1.out 2
#4 smtp_error_c <= #1.out 3
#5 smtp_error_t <= #1.out 4
_END_CFC_
END_PROGRAM

(* POU SPIDER_DEMO, CFC *)
PROGRAM SPIDER_DEMO
VAR
	SPIDER_ACCESS: SPIDER_ACCESS;
	IP_CONTROL: IP_CONTROL;
	S_BUF: NETWORK_BUFFER;
	R_BUF: NETWORK_BUFFER;
	MODE: BYTE := 1;
	IP_C: IP_C;
	VALUE: STRING;
	VAR_NAME: STRING(40) := 'RTC_SECONDS';
	ERROR: DWORD;
END_VAR
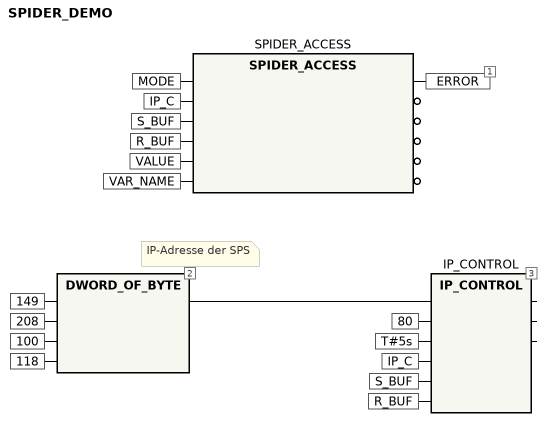
_CFC_ (* Continuous Function Chart, elements in execution order *)
#0 SPIDER_ACCESS:SPIDER_ACCESS(MODE, IP_C, S_BUF, R_BUF, VALUE, VAR_NAME)
#1 ERROR <= #0.out 1
#2 DWORD_OF_BYTE(149, 208, 100, 118)
#3 IP_CONTROL:IP_CONTROL(#2, 80, T#5s, IP_C, S_BUF, R_BUF)
(* IP-Adresse der SPS *)
_END_CFC_
END_PROGRAM

(* POU SPIDER_ACCESS, ST *)
FUNCTION_BLOCK SPIDER_ACCESS
VAR_IN_OUT
	IP_C : IP_C;(*IP_Control Verwaltungsstruktur*)
	S_BUF : NETWORK_BUFFER;
	R_BUF : NETWORK_BUFFER;
	VALUE : STRING;
	VAR_NAME : STRING(40);
END_VAR
VAR_INPUT
	MODE : BYTE;
END_VAR
VAR_OUTPUT
	ERROR : DWORD;
END_VAR
VAR
	state : INT;
	st_tmp : STRING(STRING_LENGTH);
	URL_DATA : url;
	HTTP_GET : HTTP_GET;
	value_len :	UINT;
	body_len :	UINT;
	mode_save : BYTE;
END_VAR

(*
version 1.1	12. apr. 2011
programmer 	ks
tested by		ks
*)
CASE state OF

00:
	IF MODE > BYTE#0 AND MODE < BYTE#3 THEN
		MODE_SAVE := MODE; (* Modus speichern *)
		(* wenn kein '.' in Name dann ist es eine globale variable *)
		IF FIND(VAR_NAME,'.') = 0 THEN
			st_tmp := CONCAT('%40GV.',VAR_NAME);
		ELSE
			st_tmp := VAR_NAME;
		END_IF;

		IF MODE_SAVE = BYTE#2 THEN (* 2 = Write *)
			VALUE_LEN := INT_TO_UINT(LEN(VALUE));
			st_tmp := CONCAT(st_tmp,'+');
			st_tmp := CONCAT(st_tmp,VALUE);
			URL_DATA:=STRING_TO_URL(STR:= CONCAT('http://x/dir/cgi-bin/writeVal.exe?',st_tmp),DEFAULT_PROTOCOL:='',DEFAULT_PATH:='');
		ELSE
			URL_DATA:=STRING_TO_URL(STR:= CONCAT('http://x/dir/cgi-bin/readVal.exe?',st_tmp),DEFAULT_PROTOCOL:='',DEFAULT_PATH:='');
		END_IF;

		state := 60;
	END_IF;
60:
	IF HTTP_GET.DONE THEN
		IF MODE_SAVE = BYTE#2 THEN (* Write *)
			BODY_LEN := HTTP_GET.BODY_STOP - HTTP_GET.BODY_START + BOOL_TO_UINT(HTTP_GET.BODY_STOP > UINT#0);
			ERROR := BOOL_TO_DWORD(BODY_LEN <> VALUE_LEN);
		ELSE (* Read *)
			IF HTTP_GET.BODY_START > 0 THEN
				VALUE := BUFFER_TO_STRING(PT:=ADR(R_BUF.BUFFER),SIZE:=R_BUF.SIZE,START:=UINT_TO_INT(HTTP_GET.BODY_START),STOP:=UINT_TO_INT(HTTP_GET.BODY_STOP));
			ELSE
				VALUE := '';
			END_IF;
		END_IF;
		STATE   := 100;

	ELSIF (HTTP_GET.ERROR > DWORD#00) THEN
		ERROR := HTTP_GET.ERROR;
		STATE   := 100;
	END_IF;

100:
	(* UNLOCK HTTP DATA *)
	IF HTTP_GET.DONE = FALSE THEN
		STATE := 0;
	END_IF;

END_CASE;

(* HTTP_GET *)
HTTP_GET(	IP_C:=IP_C,
			S_BUF:=S_BUF,
			R_BUF:=R_BUF,
			IP4:=DWORD#00,
			GET:=state=60,
			MODE:=BYTE#0,
			UNLOCK_BUF:=state=100,
			URL_DATA:=URL_DATA
			);

(* revision history
ks	18. mar. 2009	rev 1.0
	original version

ks	12. apr. 2011	rev 1.1
	fehlerkorrektur bei buffer_to_string
*)
END_FUNCTION_BLOCK

(* POU TELNET_LOG_DEMO, CFC *)
PROGRAM TELNET_LOG_DEMO
VAR
	TELNET_LOG: TELNET_LOG;
	IPC: IP_C;
	S_BUF: NETWORK_BUFFER;
	R_BUF: NETWORK_BUFFER;
	READY: BOOL;
	IP_CONTROL: IP_CONTROL;
	TON_1: TON;
	LOG_MSG: LOG_MSG;
END_VAR
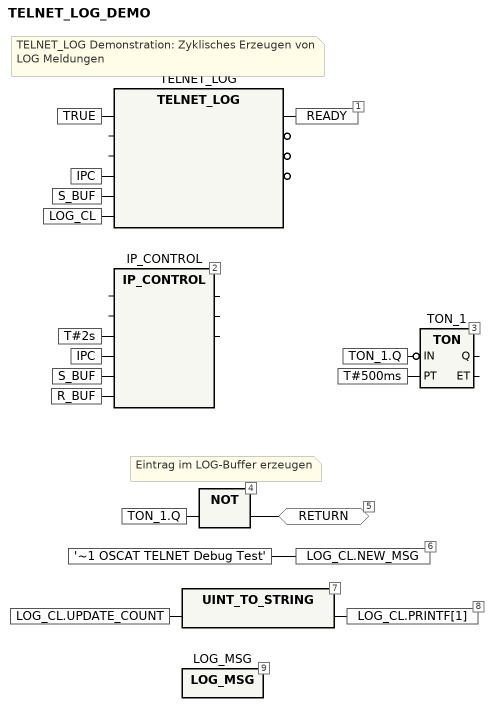
_CFC_ (* Continuous Function Chart, elements in execution order *)
#0 TELNET_LOG:TELNET_LOG(TRUE, -, -, IPC, S_BUF, LOG_CL)
#1 READY <= #0.out 1
#2 IP_CONTROL:IP_CONTROL(-, -, T#2s, IPC, S_BUF, R_BUF)
#3 TON_1:TON(IN: NOT TON_1.Q, PT: T#500ms)
#4 NOT(TON_1.Q)
#5 <RETURN> <= #4
#6 LOG_CL.NEW_MSG <= '~1 OSCAT TELNET Debug Test'
#7 UINT_TO_STRING(LOG_CL.UPDATE_COUNT)
#8 LOG_CL.PRINTF[1] <= #7
#9 LOG_MSG:LOG_MSG()
(* Eintrag im LOG-Buffer erzeugen *)
(* TELNET_LOG Demonstration: Zyklisches Erzeugen von LOG Meldungen *)
_END_CFC_
END_PROGRAM

(* POU TELNET_LOG, ST *)
FUNCTION_BLOCK TELNET_LOG
VAR_IN_OUT
	IP_C : IP_C;
	S_BUF : NETWORK_BUFFER;
	LOG_CL : LOG_CONTROL;
END_VAR
VAR_INPUT
	ENABLE : BOOL;
	OPTION : BYTE := BYTE#2#1000_1100; (* no flush buffer (7) , CR&LF (3), Colors (2), AUTOWRAP (1), Screen-Init (0) *)
	PORT : WORD := 23; (* Port Nummer *)
END_VAR
VAR_OUTPUT
	READY : BOOL;
END_VAR
VAR
	TELNET_PRINT : TELNET_PRINT;
	done : BOOL;
	init : BOOL;
	watchdog : TON;
	ci : INT;
	pi : INT;
	pi_last : INT;
	send : BOOL;
END_VAR

(*
version 1.1	03. Dec. 2011
programmer 	ks
tested BY	ks

TELNET_LOG sendet alle Texte vom LOG_BUFFER an eine TELNET_Konsole
*)
IF NOT init THEN
	init := TRUE;
	IF OPTION > 0 THEN
		TELNET_PRINT.OPTION := OPTION;
	END_IF;
	IF PORT > 0 THEN (* bei portvorgabe wird der standardport überschrieben *)
		TELNET_PRINT.PORT := PORT;
	END_IF;
  	WATCHDOG.PT := T#1ms;
END_IF;

WATCHDOG(IN:=FALSE); (* Timer stoppen *)

ci := LOG_CL.IDX;

(* CONNECT_OFF Flanke auswerten *)
IF IP_C.C_STATE = BYTE#1 THEN
	pi := 0;
	init := FALSE;
END_IF;

REPEAT
	IF pi <> ci AND IP_C.C_STATE > BYTE#127 THEN
		IF pi = 0 AND LOG_CL.RING_MODE THEN pi := ci; END_IF;
		pi_last := pi;
		pi := pi + 1;
		IF pi > LOG_CL.SIZE THEN pi := 1; END_IF;
		SEND := TRUE;
	ELSE
		SEND := FALSE;
	END_IF;

	TELNET_PRINT(	IP_C := IP_C,
					S_BUF := S_BUF,
					ENABLE := ENABLE,
					SEND := SEND,
					TEXT := LOG_CL.MSG[pi],
					BACK_COLOR := DWORD_TO_BYTE(SHL(LOG_CL.MSG_OPTION[pi],8)),
					FRONT_COLOR := DWORD_TO_BYTE(LOG_CL.MSG_OPTION[pi] ));
	READY := TELNET_PRINT.READY;
	done := TELNET_PRINT.DONE;

	IF SEND AND NOT done THEN
		pi := pi_last;
	END_IF;

	WATCHDOG(IN:=TRUE);

UNTIL (WATCHDOG.Q OR NOT done )
END_REPEAT;

(* revision history
ks	14. aug. 2009	rev 1.0
	original version

ks	03. dec. 2011	rev 1.1
	neue parameter und initialisierung optimiert

*)
END_FUNCTION_BLOCK

(* POU TELNET_PRINT, ST *)
FUNCTION_BLOCK TELNET_PRINT
VAR_IN_OUT
	IP_C : IP_C;
	S_BUF : NETWORK_BUFFER;
END_VAR
VAR_INPUT
	TEXT : STRING(STRING_LENGTH);
	ENABLE : BOOL;
	SEND : BOOL;
	OPTION : BYTE := BYTE#2#1000_1100; (* no flush buffer (7) , CR&LF (3), Colors (2), AUTOWRAP (1), Screen-Init (0) *)
	BACK_COLOR : BYTE;
	FRONT_COLOR : BYTE;
	X_POS : BYTE;
	Y_POS : BYTE;
	PORT : WORD := 23; (* Port Nummer *)
END_VAR
VAR_OUTPUT
	READY : BOOL;
	DONE : BOOL;
END_VAR
VAR
	last_fc : BYTE;
	state : INT;
	x : INT := -1;
	ip_state : BYTE;
	ip_id : BYTE;
	IP_FIFO : IP_FIFO;
	init : BOOL;
	b0_screen_clear : BOOL;
	b1_autowrap : BOOL;
	b2_color : BOOL;
	b3_cr_lr : BOOL;
	b7_no_flush : BOOL;
END_VAR

(*
version 1.4		03. dec. 2011
programmer 		ks
tested by			ks

TELNET_PRINT sendet einem TEXT in Farbe an Position X,Y an eine TELNET-Konsole
*)
READY := IP_C.C_STATE > BYTE#127;
DONE := FALSE;

CASE state OF

00: (* Warten auf Freigabe *)
	IF ENABLE THEN
		state := 10;
		ip_state := BYTE#1; (* Anmelden *)
	END_IF;

10: (* Bei IP_Control anmelden und auf freigabe warten *)
	IF ip_state = BYTE#3 THEN

		(* IP Datenverkehr einrichten *)
		IP_C.C_PORT := PORT; (* Portnummer eintragen *)
		IP_C.C_IP := DWORD#00; (* IP eintragen *)
		IP_C.C_MODE := BYTE#4; (* Mode: TCP+PASSIV+PORT *)
		IP_C.TIME_RESET := TRUE; (* Zeitueberwachung rücksetzen *)
		IP_C.C_ENABLE := TRUE; (* Verbindungsaufbau freigeben *)
		IP_C.R_OBSERVE := FALSE; (* keine Empfangsueberwachung *)
		state := 20;
	END_IF;

20:	IF IP_C.ERROR > DWORD#0 THEN
		IP_C.TIME_RESET := TRUE; (* Fehler rücksetzen *)
	END_IF;
	IF S_BUF.SIZE = UINT#0 THEN (* Datensenden nicht aktiv *)
		IF NOT ENABLE THEN
			ip_state := BYTE#4; (* Verbindung abbauen - Ressource freigeben *)
			IP_C.C_ENABLE := FALSE; (* Verbindungsabbau *)
			state := 0;
		END_IF;
		IF IP_C.C_STATE = BYTE#1 THEN (* positive Flanke Connect off *)
			init := FALSE;
		ELSIF READY THEN (* Verbindung vorhanden *)
			IF IP_C.C_STATE = BYTE#254 AND NOT INIT THEN (* positive Flanke Connect on *)
				(* Var Init ist notwendig, damit der Baustein im selben zyklus mehrmals ausgerufen werden kann *)
				init := TRUE;
				b0_screen_clear := (OPTION AND BYTE#2#0000_0001) > BYTE#0;
				b1_autowrap := (OPTION AND BYTE#2#0000_0010) > BYTE#0;
				b2_color := (OPTION AND BYTE#2#0000_0100) > BYTE#0;
				b3_cr_lr := (OPTION AND BYTE#2#0000_1000) > BYTE#0;
				b7_no_flush := (OPTION AND BYTE#2#1000_0000) > BYTE#0;

				last_fc := NOT FRONT_COLOR; (* aktualisierung der Farben erzwingen !*)
				x := 0;

				(* AUTOWRAP OFF/ON *)
				S_BUF.BUFFER[x] := BYTE#16#1B; (* ESC *)
				x := x +1;
				S_BUF.BUFFER[x] := BYTE#16#5B; (* [ *)
				x := x +1;
				S_BUF.BUFFER[x] := BYTE#16#3F; (* ? *)
				x := x +1;
				S_BUF.BUFFER[x] := BYTE#16#37; (* 7 *)
				x := x +1;
				S_BUF.BUFFER[x] := SEL(b1_autowrap, BYTE#16#6C (* l *),BYTE#16#68 (* h *));

				IF b0_screen_clear THEN
					IF b2_color THEN
						x := x +1;
						S_BUF.BUFFER[x] := BYTE#16#1B; (* ESC *)
						x := x +1;
						S_BUF.BUFFER[x] := BYTE#16#5B; (* [ *)
						x := x +1;
						S_BUF.BUFFER[x] := BYTE#16#30; (* 0 *)
						x := x +1;
						S_BUF.BUFFER[x] := BYTE#16#3B; (* ; *)
						x := x +1;
						S_BUF.BUFFER[x] := BYTE#16#33; (* 3 *)
						x := x +1;
						S_BUF.BUFFER[x] := (FRONT_COLOR AND BYTE#2#00000111) OR BYTE#16#30; (* Einerstelle Farbe Foreground ausgeben *)
						x := x +1;
						S_BUF.BUFFER[x] := BYTE#16#3B; (* ; *)
						x := x +1;
						S_BUF.BUFFER[x] := BYTE#16#34; (* 4 *)
						x := x +1;
						S_BUF.BUFFER[x] := (BACK_COLOR AND BYTE#2#00000111) OR BYTE#16#30; (* Einerstelle Farbe Background ausgeben *)
						x := x +1;
						S_BUF.BUFFER[x] := BYTE#16#6D; (* m *)
					END_IF;
					(* Screen Clear *)
					x := x +1;
					S_BUF.BUFFER[x] := BYTE#16#1B; (* ESC *)
					x := x +1;
					S_BUF.BUFFER[x] := BYTE#16#5B; (* [ *)
					x := x +1;
					S_BUF.BUFFER[x] := BYTE#16#32; (* 2 *)
					x := x +1;
					S_BUF.BUFFER[x] := BYTE#16#4A; (* J *)
				ELSE
					x := x +1;
					S_BUF.BUFFER[x] := BYTE#16#0A; (* neue Zeile *)
				END_IF;
			END_IF;

			(* buffer voll , oder Daten sind vorhanden und kein weiterer Sendewunsch *)
			IF (INT_TO_UINT(x + LEN(TEXT) + 21) > SIZEOF(S_BUF.BUFFER)) OR (x >= 0 AND NOT SEND) THEN
				S_BUF.SIZE := INT_TO_UINT(x + 1); (* Länge eintragen -> Datensenden starten *)
				x := -1;
			ELSIF SEND THEN

				(* aktuelle Farbe bestimmen  *)
				IF b2_color AND FRONT_COLOR <> last_FC THEN
					(* Farbeinstellung: ANSI-Sequenz ESC[X;Y;Zm ausgeben *)
					x := x + 1;
					S_BUF.BUFFER[x] := BYTE#16#1B; (* ESC *)
					x := x + 1;
					S_BUF.BUFFER[x] := BYTE#16#5B; (* [ *)
					(* Farbeinstellung: dunkel oder Hell und blinken bestimmen *)
					IF ((FRONT_COLOR AND BYTE#2#0001_1000) XOR (last_FC AND BYTE#2#0001_1000)) <> BYTE#00 OR TRUE THEN
						x := x + 1;
						S_BUF.BUFFER[x] := BYTE#16#30; (* 0  *)
						x := x + 1;
						S_BUF.BUFFER[x] := BYTE#16#3B; (* ; *)
						(* keine dunklen Farben gewünscht -> dann Bold & Bright *)
						IF (FRONT_COLOR AND BYTE#2#00001000) = BYTE#0 THEN
							(* auf Bold & Bright Farben umstellen *)
							x := x + 1;
							S_BUF.BUFFER[x] := BYTE#16#31; (* 1 *)
							x := x + 1;
							S_BUF.BUFFER[x] := BYTE#16#3B; (* ; *)
						END_IF;
						(* blinkenden Farben gewünscht *)
						IF (FRONT_COLOR AND BYTE#2#00010000) > BYTE#0 THEN
							(* auf Blinkenden Farbe umstellen *)
							x := x + 1;
							S_BUF.BUFFER[x] := BYTE#16#35; (* 5 *)
							x := x + 1;
							S_BUF.BUFFER[x] := BYTE#16#3B; (* ; *)
						END_IF;
					END_IF;
					(* Zehnerstelle Farbe Foreground ausgeben *)
					x := x + 1;
					S_BUF.BUFFER[x] := BYTE#16#33; (* 3 *)
					(* Einerstelle Farbe Foreground ausgeben *)
					x := x + 1;
					S_BUF.BUFFER[x] := (FRONT_COLOR AND BYTE#2#00000111) OR BYTE#16#30;
					x := x + 1;
					S_BUF.BUFFER[x] := BYTE#16#6D; (* m *)
					(* neue Farbe als letzt verwendete speichern *)
					last_FC := FRONT_COLOR;
				END_IF;

				(* Cursor positionieren *)
				IF X_POS > BYTE#0 AND Y_POS > BYTE#0 THEN
					x := x + 1;
					S_BUF.BUFFER[x] := BYTE#16#1B; (* ESC *)
					x := x + 1;
					S_BUF.BUFFER[x] := BYTE#16#5B; (* [ *)
					(* Zehnerstelle Y_POS ausgeben *)
					x := x + 1;
					S_BUF.BUFFER[x] := SHR(INT_TO_BCDC(BYTE_TO_INT(Y_POS)),4) OR BYTE#16#30;
					(* Einerstelle Y_POS ausgeben *)
					x := x + 1;
					S_BUF.BUFFER[x] := (INT_TO_BCDC(BYTE_TO_INT(Y_POS)) AND BYTE#16#0F) OR BYTE#16#30;
					x := x + 1;
					S_BUF.BUFFER[x] := BYTE#16#3B; (* ; *)
					(* Zehnerstelle X_POS ausgeben *)
					x := x + 1;
					S_BUF.BUFFER[x] := SHR(INT_TO_BCDC(BYTE_TO_INT(X_POS)),4) OR BYTE#16#30;
					(* Einerstelle X_POS ausgeben *)
					x := x + 1;
					S_BUF.BUFFER[x] := (INT_TO_BCDC(BYTE_TO_INT(X_POS)) AND BYTE#16#0F) OR BYTE#16#30;
					x := x + 1;
					S_BUF.BUFFER[x] := BYTE#16#48; (* H *)
				END_IF;

				(* text ausgeben *)
				IF LEN(TEXT) > 0 THEN
					_STRING_TO_BUFFER(str:=TEXT,pos:=x + 1,pt :=ADR(S_BUF.BUFFER), size:=SIZEOF(S_BUF.BUFFER));
					x := x + LEN(TEXT);
				END_IF;

				IF b3_cr_lr THEN (* Option: CR,LF ausgeben *)
					x := x + 1;
					S_BUF.BUFFER[x] := BYTE#16#0D;
					x := x + 1;
					S_BUF.BUFFER[x] := BYTE#16#0A;
				END_IF;

				DONE := TRUE; (* Fertig in Buffer eingetragen *)

				IF b7_no_flush THEN (* Option: no buffer flush *)
					(* buffer sofort senden - aktuellen Schreibindex speichern -> Senden anstossen *)
					S_BUF.SIZE := INT_TO_UINT(x + 1);
					x := -1;
				END_IF;
			END_IF;
		END_IF;
	END_IF;
END_CASE;

(* IP_FIFO *)
IP_FIFO(FIFO:=IP_C.FIFO,STATE:=ip_state,ID:=ip_id);

(* revision history
ks	05. jan. 2009	rev 1.0
	original version

ks	20. oct. 2009	rev 1.1
	Networkbuffer und Buffer-funktionen auf Basis 0

ks	20. oct. 2009	rev 1.2
	STRING(STRING_LENGTH)

ks	17. may. 2011	rev 1.3
	automatischer re-connect

ks	03. dec. 2011	rev 1.4
	initialisierung verbessert, Port Nummer als Parmeter

*)
END_FUNCTION_BLOCK

(* POU LOG_MSG, ST *)
FUNCTION_BLOCK LOG_MSG
(* VAR_EXTERNAL
	LOG_CL :	LOG_CONTROL;
END_VAR *)
VAR
	FB_PRINT_SF :PRINT_SF;
	idX : INT;
END_VAR

(*
version 1.0		01 mai 2010
programmer		ks
tested by		ks

LOG_MSG trägt Meldungen in den Loggingbuffer ein
*)
IF DWORD_TO_BYTE(SHL(LOG_CL.NEW_MSG_OPTION,16)) > LOG_CL.LEVEL THEN RETURN; END_IF; (* Logging freigegeben ?*)

FB_PRINT_SF(PRINTF_DATA := LOG_CL.PRINTF,STR := LOG_CL.NEW_MSG);

IF LOG_CL.RESET THEN (* Logeinträge löschen *)
	LOG_CL.RESET := FALSE;
	LOG_CL.RING_MODE := FALSE;
	LOG_CL.IDX := 0;
	LOG_CL.UPDATE_COUNT := LOG_CL.UPDATE_COUNT + UINT#1; (* UpdateCount erhöhen *)
END_IF;

IF LOG_CL.SIZE > 0 THEN (* size wert ist eingetragen *)
	IF LEN(LOG_CL.NEW_MSG) > 0 THEN (* Meldung in Puffer eintragen *)
		IF (LOG_CL.IDX >= LOG_CL.SIZE) THEN
			LOG_CL.RING_MODE := TRUE; (* bei Überlauf = Ringbuffermodus *)
			LOG_CL.IDX := 0; (* wieder auf arrayanfang positionieren *)
		END_IF;

		LOG_CL.UPDATE_COUNT := LOG_CL.UPDATE_COUNT + UINT#1; (* UpdateCount erhöhen *)
		LOG_CL.IDX := LOG_CL.IDX + INT#1; (* nächste freie Position *)
		idx := LOG_CL.IDX; (* lade aktuelle Log-Puffer Positition *)
		LOG_CL.MSG[idx] := LOG_CL.NEW_MSG; (* neuen Log-String in puffer ablegen  *)
		LOG_CL.MSG_OPTION[idx] := LOG_CL.NEW_MSG_OPTION; (* neue Log-String Option in puffer ablegen  *)
		LOG_CL.NEW_MSG := ''; (* letzten Log-String löschen *)
	END_IF;
END_IF;
END_FUNCTION_BLOCK

(* POU PRINT_SF, ST *)
FUNCTION_BLOCK PRINT_SF
VAR_IN_OUT
	PRINTF_DATA : PRINTF_DATA;
	STR : STRING(LOG_SIZE);
END_VAR
VAR
	pos : INT;
	c : INT;
	src : STRING(1) := '~';
	run : BOOL;
END_VAR

(*

version 1.0 		14. aug. 2009
programmer 	ks
tested by		ks

PRINTF erzeugt aus einem Parameterstring und den übergebenen Parameterdaten einen Text
*)
IF LEN(STR) > 0 THEN
	run := TRUE;

	WHILE (run) DO
		pos := FIND(STR,src);
		PRINTF_DATA[10] := '';

		IF pos = 0 THEN
			run:= FALSE;
		ELSE
			c := CODE(STR:=STR,POS:=pos + 1);
			IF ISC_NUM(INT_TO_BYTE(c)) THEN
				c := c - 48; (* notwendig weil innerhalb einer indexangabe nur eine var stehen darf *)
				PRINTF_DATA[10] := PRINTF_DATA[c]; (* Kommando 1-9 ergibt Parameterindex 1-9 *)
				(* Parameter gegen Text tauschen *)
			END_IF;
			IF LEN(PRINTF_DATA[10]) + LEN(STR) > LOG_SIZE THEN
				PRINTF_DATA[10] := '..';
			END_IF;
			(* pcworx: aus und eingangsstring muss verschieden sein *)
			PRINTF_DATA[11] := STR;
			STR := REPLACE(PRINTF_DATA[11],PRINTF_DATA[10],2,pos);
		END_IF;
	END_WHILE;
END_IF;

(* revision history

ks	14. aug. 2009	rev 1.0
	original version

*)
END_FUNCTION_BLOCK

(* POU TELNET_PRINT_DEMO, CFC *)
PROGRAM TELNET_PRINT_DEMO
VAR
	COUNT_BR_1: COUNT_BR;
	READY: BOOL;
	TON_1: TON;
	TEXT: STRING;
	TEXT_ATTRIBUTE: BYTE;
	GEN_SIN_1: GEN_SIN;
	X_POS: BYTE;
	Y_POS: BYTE;
	GEN_SIN_2: GEN_SIN;
	TELNET_PRINT: TELNET_PRINT;
	DONE: BOOL;
	IP_C: IP_C;
	S_BUF: NETWORK_BUFFER;
	IP_CONTROL: IP_CONTROL;
	R_BUF: NETWORK_BUFFER;
END_VAR
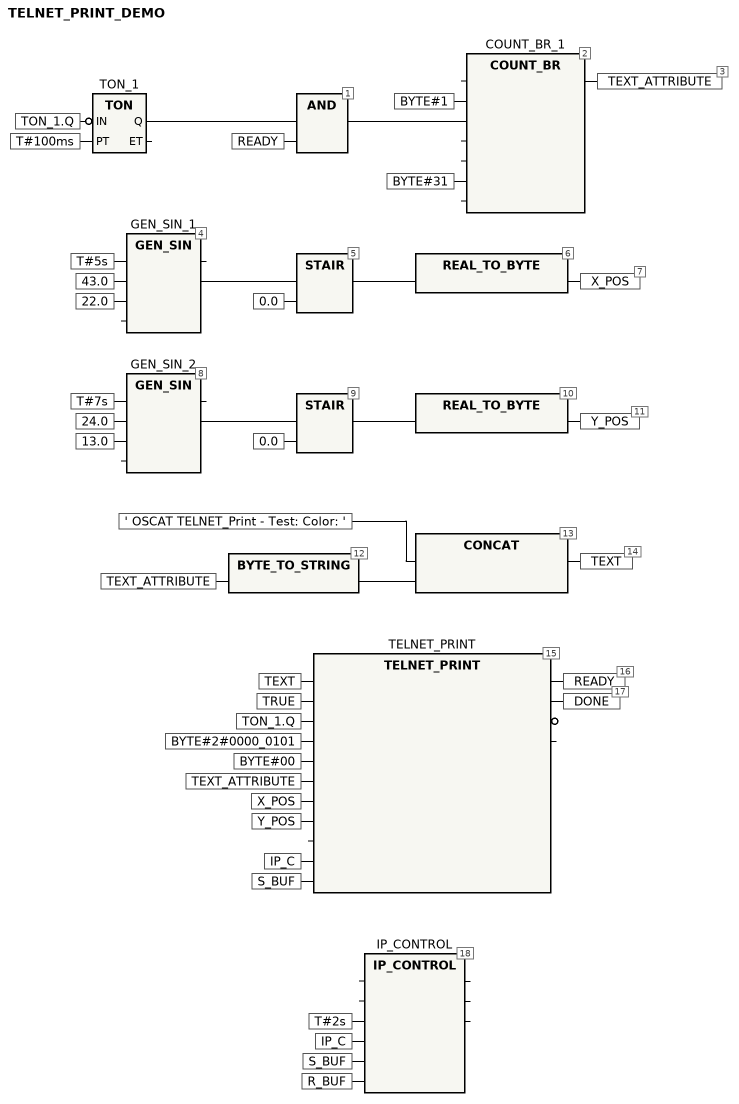
_CFC_ (* Continuous Function Chart, elements in execution order *)
#0 TON_1:TON(IN: NOT TON_1.Q, PT: T#100ms)
#1 AND(#0.Q, READY)
#2 COUNT_BR_1:COUNT_BR(-, BYTE#1, #1, -, -, BYTE#31, -)
#3 TEXT_ATTRIBUTE <= #2
#4 GEN_SIN_1:GEN_SIN(T#5s, 43.0, 22.0, -)
#5 STAIR(#4.out 2, 0.0)
#6 REAL_TO_BYTE(#5)
#7 X_POS <= #6
#8 GEN_SIN_2:GEN_SIN(T#7s, 24.0, 13.0, -)
#9 STAIR(#8.out 2, 0.0)
#10 REAL_TO_BYTE(#9)
#11 Y_POS <= #10
#12 BYTE_TO_STRING(TEXT_ATTRIBUTE)
#13 CONCAT(' OSCAT TELNET_Print - Test: Color: ', #12)
#14 TEXT <= #13
#15 TELNET_PRINT:TELNET_PRINT(TEXT, TRUE, TON_1.Q, BYTE#2#0000_0101, BYTE#00, TEXT_ATTRIBUTE, X_POS, Y_POS, -, IP_C, S_BUF)
#16 READY <= #15.out 1
#17 DONE <= #15.out 2
#18 IP_CONTROL:IP_CONTROL(-, -, T#2s, IP_C, S_BUF, R_BUF)
_END_CFC_
END_PROGRAM

(* POU TN_VISION_DEMO_1, ST *)
PROGRAM TN_VISION_DEMO_1
VAR
	FB_TN_FRAMEWORK : TN_FRAMEWORK;
	FB_LOG_MESSAGE : LOG_MSG;
	FB_LOG_VIEWPORT : LOG_VIEWPORT;
	FB_TN_SC_LINE : TN_SC_LINE;
	FB_TN_SC_FILL : TN_SC_FILL;
	FB_TN_SC_WRITE_C : TN_SC_WRITE_C;
	FB_TN_SC_BOX : TN_SC_BOX;
	FB_TN_SC_ADD_SHADOW : TN_SC_ADD_SHADOW;
	FB_TN_SC_WRITE : TN_SC_WRITE;
	FB_TN_SC_VIEWPORT : TN_SC_VIEWPORT;
	Xus_TN_MENU : us_TN_MENU;
	Xus_TN_INPUT_CONTROL : us_TN_INPUT_CONTROL;
	Xus_TN_SCREEN : us_TN_SCREEN;
	us_LOG_VIEWPORT : us_LOG_VIEWPORT;
	S_BUF : NETWORK_BUFFER;
	R_BUF : NETWORK_BUFFER;
	IP_C : IP_C;
	Gst_SysLog_Command : STRING;
	in_index : INT;
END_VAR
FB_TN_FRAMEWORK(
					us_TN_INPUT_CONTROL := Xus_TN_INPUT_CONTROL ,
					us_TN_SCREEN := Xus_TN_SCREEN ,
					us_TN_MENU := Xus_TN_MENU ,
					S_BUF := S_BUF ,
					R_BUF:= R_BUF ,
					IP_C:= IP_C ,
					PORT := WORD#0
					 );

(* Modaler Dialog aktiv ? *)
IF (Xus_TN_SCREEN.bo_Modal_Dialog = TRUE) THEN RETURN; END_IF;

IF Xus_TN_MENU.in_Menu_Selected > 0 THEN

	CASE Xus_TN_MENU.in_Menu_Selected OF

	41: (* Seite LOGIN aufrufen *)
		Xus_TN_SCREEN.in_Page_Number := INT#00;
		(* Gedächtnis löschen *)
		Xus_TN_MENU.bo_Destroy := TRUE;

	END_CASE;

	(* Echo Menu-Auswahl *)
	Gst_SysLog_Command := CONCAT('MENU_SELECT: ',INT_TO_STRING(Xus_TN_MENU.in_Menu_Selected));

	(* Menu-Auswahl löschen *)
	Xus_TN_MENU.in_Menu_Selected := 0;

END_IF;

(* Initialisierung der Daten und Strukturen *)
IF (Xus_TN_SCREEN.in_Page_Number = INT#00 ) THEN
	Xus_TN_SCREEN.in_Page_Number := INT#01;

	(* Clear-Screen (Farbe setzen + Display löschen) *)
	Xus_TN_SCREEN.by_Clear_Screen_Attr := BYTE#16#00;
	Xus_TN_SCREEN.bo_Clear_Screen := TRUE;

	(* Screen initialisieren (mit Leerzeichen füllen) *)
	FB_TN_SC_FILL(	Iin_X1 := INT#00,
					Iin_Y1 := INT#00,
					Iin_X2 := INT#79,
					Iin_Y2 := INT#23,
					Iby_CHAR := BYTE#179,
					Iby_Attr := BYTE#16#76,
					Xus_TN_SCREEN := Xus_TN_SCREEN);

	(* Titlezeile zeichnen *)
	FB_TN_SC_FILL(	Iin_X1 := INT#00,
					Iin_Y1 := INT#00,
					Iin_X2 := INT#79,
					Iin_Y2 := INT#00,
					Iby_CHAR := BYTE#32,
					Iby_Attr := BYTE#16#07,
					Xus_TN_SCREEN := Xus_TN_SCREEN);

	(* Title zeichnen *)
	FB_TN_SC_WRITE(	Iin_X := INT#00,
					Iin_Y := INT#00,
					Iby_ATTR := BYTE#16#77,
					Ist_STRING := ' TELNET-VISION BIOS v1.0',
					Xus_TN_SCREEN := Xus_TN_SCREEN);

	(* Fusszeile zeichnen *)
	FB_TN_SC_FILL(	Iin_X1 := INT#00,
					Iin_Y1 := INT#23,
					Iin_X2 := INT#79,
					Iin_Y2 := INT#23,
					Iby_CHAR := BYTE#32,
					Iby_Attr := BYTE#16#37,
					Xus_TN_SCREEN := Xus_TN_SCREEN);

	(* Rahmen für Viewport zeichnen *)
	FB_TN_SC_BOX(	Iin_X1 := INT#03,
					Iin_Y1 := INT#03,
					Iin_X2 := INT#75,
					Iin_Y2 := INT#19,
					Iby_FILL := BYTE#16#20, (* Füllung *)
					Iin_BORDER := INT#02, (* Double-Line Border *)
					Iby_ATTR := BYTE#16#74, (* Weiss , Blau *)
					Xus_TN_SCREEN := Xus_TN_SCREEN);

	(* Shadow für Rahmen von Viewport zeichnen *)
	FB_TN_SC_ADD_SHADOW(	Iin_X1 := INT#04,
							Iin_Y1 := INT#04,
							Iin_X2 := INT#76,
							Iin_Y2 := INT#20,
							Iin_OPTION := INT#00,
							Xus_TN_SCREEN := Xus_TN_SCREEN);

	(* Title Viewport zeichnen *)
	FB_TN_SC_WRITE(	Iin_X := INT#31,
					Iin_Y := INT#03,
					Iby_ATTR := BYTE#16#74,
					Ist_STRING := '[ LOGIN-DIALOG ]',
					Xus_TN_SCREEN := Xus_TN_SCREEN);

	(* LOGO Zeilen zeichnen *)
	FOR in_index := 5 TO 16 DO

		CASE in_index OF

		05: FB_TN_SC_WRITE.Ist_STRING := 'ÛÛÛÛÛÛÛÛ» ÛÛÛÛÛÛÛ» ÛÛ»      ÛÛÛ»   ÛÛ» ÛÛÛÛÛÛÛ» ÛÛÛÛÛÛÛÛ»';
		06: FB_TN_SC_WRITE.Ist_STRING := 'ÈÍÍÛÛÉÍÍ¼ ÛÛÉÍÍÍÍ¼ ÛÛº      ÛÛÛÛ»  ÛÛº ÛÛÉÍÍÍÍ¼ ÈÍÍÛÛÉÍÍ¼';
		07: FB_TN_SC_WRITE.Ist_STRING := '   ÛÛº    ÛÛÛÛÛ»   ÛÛº      ÛÛÉÛÛ» ÛÛº ÛÛÛÛÛ»      ÛÛº';
		08: FB_TN_SC_WRITE.Ist_STRING := '   ÛÛº    ÛÛÉÍÍ¼   ÛÛº      ÛÛºÈÛÛ»ÛÛº ÛÛÉÍÍ¼      ÛÛº';
		09: FB_TN_SC_WRITE.Ist_STRING := '   ÛÛº    ÛÛÛÛÛÛÛ» ÛÛÛÛÛÛÛ» ÛÛº ÈÛÛÛÛº ÛÛÛÛÛÛÛ»    ÛÛº';
		10: FB_TN_SC_WRITE.Ist_STRING := '   ÈÍ¼    ÈÍÍÍÍÍÍ¼ ÈÍÍÍÍÍÍ¼ ÈÍ¼  ÈÍÍÍ¼ ÈÍÍÍÍÍÍ¼    ÈÍ¼';
		11: FB_TN_SC_WRITE.Ist_STRING := '     ÛÛ»   ÛÛ» ÛÛ» ÛÛÛÛÛÛÛ» ÛÛ»  ÛÛÛÛÛÛ»  ÛÛÛ»   ÛÛ»';
		12: FB_TN_SC_WRITE.Ist_STRING := '     ÛÛº   ÛÛº ÛÛº ÛÛÉÍÍÍÍ¼ ÛÛº ÛÛÉÍÍÍÛÛ» ÛÛÛÛ»  ÛÛº';
		13: FB_TN_SC_WRITE.Ist_STRING := '     ÛÛº   ÛÛº ÛÛº ÛÛÛÛÛÛÛ» ÛÛº ÛÛº   ÛÛº ÛÛÉÛÛ» ÛÛº';
		14: FB_TN_SC_WRITE.Ist_STRING := '     ÈÛÛ» ÛÛÉ¼ ÛÛº ÈÍÍÍÍÛÛº ÛÛº ÛÛº   ÛÛº ÛÛºÈÛÛ»ÛÛº';
		15: FB_TN_SC_WRITE.Ist_STRING := '      ÈÛÛÛÛÉ¼  ÛÛº ÛÛÛÛÛÛÛº ÛÛº ÈÛÛÛÛÛÛÉ¼ ÛÛº ÈÛÛÛÛº';
		16: FB_TN_SC_WRITE.Ist_STRING := '       ÈÍÍÍ¼   ÈÍ¼ ÈÍÍÍÍÍÍ¼ ÈÍ¼  ÈÍÍÍÍÍ¼  ÈÍ¼  ÈÍÍÍ¼';

		END_CASE;

		FB_TN_SC_WRITE(	Iin_Y := in_index,
						Iin_X := INT#11,
						Iby_ATTR := BYTE#16#34,
						Xus_TN_SCREEN := Xus_TN_SCREEN);
	END_FOR;

	(* Trennlinie zeichnen *)
	FB_TN_SC_LINE(	Iin_X1 := INT#03,
					Iin_Y1 := INT#17,
					Iin_X2 := INT#75,
					Iin_Y2 := INT#17,
					Iby_ATTR := BYTE#16#74,
					Iby_BORDER := BYTE#02,
					Xus_TN_SCREEN := Xus_TN_SCREEN);

	(* Alle Input-Controls initialisieren *)

	Xus_TN_INPUT_CONTROL.bo_Enable := FALSE;

	(* Initialisierung der Eingabe-Zeile *)
	Xus_TN_INPUT_CONTROL.usa_TN_INPUT_CONTROL_DATA[1].in_Type := INT#01;
	Xus_TN_INPUT_CONTROL.usa_TN_INPUT_CONTROL_DATA[1].in_Y := INT#18;
	Xus_TN_INPUT_CONTROL.usa_TN_INPUT_CONTROL_DATA[1].in_X := INT#49;
	Xus_TN_INPUT_CONTROL.usa_TN_INPUT_CONTROL_DATA[1].by_Attr_mF := BYTE#16#17;
	Xus_TN_INPUT_CONTROL.usa_TN_INPUT_CONTROL_DATA[1].by_Attr_oF := BYTE#16#47;
	Xus_TN_INPUT_CONTROL.usa_TN_INPUT_CONTROL_DATA[1].in_Cursor_Pos := INT#0;
	Xus_TN_INPUT_CONTROL.usa_TN_INPUT_CONTROL_DATA[1].bo_Input_Only_Num := FALSE;
	Xus_TN_INPUT_CONTROL.usa_TN_INPUT_CONTROL_DATA[1].bo_Input_Hidden := TRUE;
	Xus_TN_INPUT_CONTROL.usa_TN_INPUT_CONTROL_DATA[1].st_Input_Mask := '                ';
	Xus_TN_INPUT_CONTROL.usa_TN_INPUT_CONTROL_DATA[1].st_Input_Data := Xus_TN_INPUT_CONTROL.usa_TN_INPUT_CONTROL_DATA[1].st_Input_Mask;
	Xus_TN_INPUT_CONTROL.usa_TN_INPUT_CONTROL_DATA[1].st_Input_ToolTip := ' enter password | press enter to login     |';
	Xus_TN_INPUT_CONTROL.usa_TN_INPUT_CONTROL_DATA[1].in_Input_Option := INT#00;
	Xus_TN_INPUT_CONTROL.usa_TN_INPUT_CONTROL_DATA[1].in_Title_Y_Offset := INT#00;
	Xus_TN_INPUT_CONTROL.usa_TN_INPUT_CONTROL_DATA[1].in_Title_X_Offset := -12;
	Xus_TN_INPUT_CONTROL.usa_TN_INPUT_CONTROL_DATA[1].by_Title_Attr := BYTE#16#34;
	Xus_TN_INPUT_CONTROL.usa_TN_INPUT_CONTROL_DATA[1].st_Title_String := 'password:  [                ]';

	(* Initialisierung Selection Text *)
	Xus_TN_INPUT_CONTROL.usa_TN_INPUT_CONTROL_DATA[2].in_Type := INT#03;
	Xus_TN_INPUT_CONTROL.usa_TN_INPUT_CONTROL_DATA[2].in_Y := INT#18;
	Xus_TN_INPUT_CONTROL.usa_TN_INPUT_CONTROL_DATA[2].in_X := INT#18;
	Xus_TN_INPUT_CONTROL.usa_TN_INPUT_CONTROL_DATA[2].by_Attr_mF := BYTE#16#17;
	Xus_TN_INPUT_CONTROL.usa_TN_INPUT_CONTROL_DATA[2].by_Attr_oF := BYTE#16#47;
	Xus_TN_INPUT_CONTROL.usa_TN_INPUT_CONTROL_DATA[2].st_Input_ToolTip := ' select user       | press enter to select |';
	Xus_TN_INPUT_CONTROL.usa_TN_INPUT_CONTROL_DATA[2].in_Input_Option := INT#00;
	Xus_TN_INPUT_CONTROL.usa_TN_INPUT_CONTROL_DATA[2].in_Title_Y_Offset := INT#00;
	Xus_TN_INPUT_CONTROL.usa_TN_INPUT_CONTROL_DATA[2].in_Title_X_Offset := INT#00;
	Xus_TN_INPUT_CONTROL.usa_TN_INPUT_CONTROL_DATA[2].by_Title_Attr := BYTE#16#34;
	Xus_TN_INPUT_CONTROL.usa_TN_INPUT_CONTROL_DATA[2].st_Title_String := ' user ';
	Xus_TN_INPUT_CONTROL.usa_TN_INPUT_CONTROL_DATA[2].st_Input_Mask := '           ';
	Xus_TN_INPUT_CONTROL.usa_TN_INPUT_CONTROL_DATA[2].st_Input_Data := 'admin#guest#maintenance';

	(* Control-Tool-Tip *)
	Xus_TN_INPUT_CONTROL.in_ToolTip_Y := INT#23;
	Xus_TN_INPUT_CONTROL.in_ToolTip_X := INT#00;
	Xus_TN_INPUT_CONTROL.by_ToolTip_Attr := BYTE#16#37;
	Xus_TN_INPUT_CONTROL.in_ToolTip_Size := INT#80;

	(* Control-Verwaltung initialisieren *)
	Xus_TN_INPUT_CONTROL.in_Count := INT#02;
	Xus_TN_INPUT_CONTROL.bo_Enable := TRUE;
	Xus_TN_INPUT_CONTROL.bo_Reset_Fokus := TRUE;

END_IF;

IF (Xus_TN_SCREEN.in_Page_Number = INT#01) THEN
	(* eingegebenen String übernehmen *)
	IF Xus_TN_INPUT_CONTROL.usa_TN_INPUT_CONTROL_DATA[1].bo_Input_Entered = TRUE THEN

		Xus_TN_INPUT_CONTROL.usa_TN_INPUT_CONTROL_DATA[1].bo_Input_Entered := FALSE;
		Xus_TN_INPUT_CONTROL.usa_TN_INPUT_CONTROL_DATA[1].st_Input_String :=
			LOWERCASE(str:=Xus_TN_INPUT_CONTROL.usa_TN_INPUT_CONTROL_DATA[1].st_Input_String);

		IF Xus_TN_INPUT_CONTROL.usa_TN_INPUT_CONTROL_DATA[1].st_Input_String = 'oscat' THEN
			Xus_TN_SCREEN.in_Page_Number := INT#10;

			Gst_SysLog_Command := CONCAT('LOGON: USER-',Xus_TN_INPUT_CONTROL.usa_TN_INPUT_CONTROL_DATA[2].st_Input_String);

		ELSE
			FB_TN_SC_WRITE_C(	Iin_X := Xus_TN_INPUT_CONTROL.in_ToolTip_X,
								Iin_Y := Xus_TN_INPUT_CONTROL.in_ToolTip_Y,
								Iby_ATTR := BYTE#16#F1,
								Iin_OPTION := INT#02, (* Center-String *)
								Iin_LENGTH := Xus_TN_INPUT_CONTROL.in_ToolTip_Size,
								Ist_STRING := 'Password Failed   ',
								Xus_TN_SCREEN := Xus_TN_SCREEN);

			Gst_SysLog_Command := CONCAT('LOGON: ',FB_TN_SC_WRITE_C.Ist_STRING);

		END_IF;
	END_IF;
END_IF;

(* Initialisierung der Daten und Strukturen *)
IF (Xus_TN_SCREEN.in_Page_Number = INT#10 ) THEN
	Xus_TN_SCREEN.in_Page_Number := INT#11;

	(* Clear-Screen (Farbe setzen + Display löschen) *)
	Xus_TN_SCREEN.by_Clear_Screen_Attr := BYTE#16#00;
	Xus_TN_SCREEN.bo_Clear_Screen := TRUE;

	(* Screen initialisieren (mit Leerzeichen füllen) *)
	FB_TN_SC_FILL(	Iin_X1 := INT#00,
					Iin_Y1 := INT#00,
					Iin_X2 := INT#79,
					Iin_Y2 := INT#23,
					Iby_CHAR := BYTE#179,
					Iby_Attr := BYTE#16#76,
					Xus_TN_SCREEN := Xus_TN_SCREEN);

	(* Titlezeile zeichnen *)
	FB_TN_SC_FILL(	Iin_X1 := INT#00,
					Iin_Y1 := INT#00,
					Iin_X2 := INT#79,
					Iin_Y2 := INT#00,
					Iby_CHAR := BYTE#32,
					Iby_Attr := BYTE#16#07,
					Xus_TN_SCREEN := Xus_TN_SCREEN);

	(* Fusszeile zeichnen *)
	FB_TN_SC_FILL(	Iin_X1 := INT#00,
					Iin_Y1 := INT#23,
					Iin_X2 := INT#79,
					Iin_Y2 := INT#23,
					Iby_CHAR := BYTE#32,
					Iby_Attr := BYTE#16#37,
					Xus_TN_SCREEN := Xus_TN_SCREEN);

	(* Rahmen für Viewport zeichnen *)
	FB_TN_SC_BOX(	Iin_X1 := INT#00,
					Iin_Y1 := INT#01,
					Iin_X2 := INT#77,
					Iin_Y2 := INT#17,
					Iby_FILL := BYTE#16#00, (* keine Füllung *)
					Iin_BORDER := INT#02, (* Double-Line Border *)
					Iby_ATTR := BYTE#16#74, (* Weiss , Blau *)
					Xus_TN_SCREEN := Xus_TN_SCREEN);

	(* Shadow für Rahmen von Viewport zeichnen *)
	FB_TN_SC_ADD_SHADOW(Iin_X1 := INT#01,
						Iin_Y1 := INT#02,
						Iin_X2 := INT#78,
						Iin_Y2 := INT#18,
						Iin_OPTION := INT#00,
						Xus_TN_SCREEN := Xus_TN_SCREEN);

	(* Trennlinie Viewport_Data und Commandline zeichnen *)
	FB_TN_SC_LINE(	Iin_X1 := INT#00,
					Iin_Y1 := INT#15,
					Iin_X2 := INT#77,
					Iin_Y2 := INT#15,
					Iby_ATTR := BYTE#16#74,
					Iby_BORDER := BYTE#02,
					Xus_TN_SCREEN := Xus_TN_SCREEN);

	(* Title Viewport zeichnen *)
	FB_TN_SC_WRITE(	Iin_X := INT#29,
					Iin_Y := INT#01,
					Iby_ATTR := BYTE#16#74,
					Ist_STRING := '[ SYSTEM-CONSOLE ]',
					Xus_TN_SCREEN := Xus_TN_SCREEN);

	(* Rahmen für Parameter-Feld zeichnen *)
	FB_TN_SC_BOX(	Iin_X1 := INT#02,
					Iin_Y1 := INT#19,
					Iin_X2 := INT#74,
					Iin_Y2 := INT#21,
					Iby_FILL := BYTE#16#20,
					Iin_BORDER := INT#01, (* Double-Line Border *)
					Iby_ATTR := BYTE#16#74, (* Weiss , Blau *)
					Xus_TN_SCREEN := Xus_TN_SCREEN);

	(* Shadow für Rahmen von Parameter-Feld zeichnen *)
	FB_TN_SC_ADD_SHADOW(Iin_X1 := INT#03,
						Iin_Y1 := INT#20,
						Iin_X2 := INT#75,
						Iin_Y2 := INT#22,
						Iin_OPTION := INT#00,
						Xus_TN_SCREEN := Xus_TN_SCREEN);

	(* Alle Input-Controls initialisieren *)

	Xus_TN_INPUT_CONTROL.bo_Enable := FALSE;

	(* Initialisierung der Eingabe-Zeile *)
	Xus_TN_INPUT_CONTROL.usa_TN_INPUT_CONTROL_DATA[1].in_Type := INT#01;
	Xus_TN_INPUT_CONTROL.usa_TN_INPUT_CONTROL_DATA[1].in_Y := INT#16;
	Xus_TN_INPUT_CONTROL.usa_TN_INPUT_CONTROL_DATA[1].in_X := INT#09;
	Xus_TN_INPUT_CONTROL.usa_TN_INPUT_CONTROL_DATA[1].by_Attr_mF := BYTE#16#72; (* Weiss, Grün *)
	Xus_TN_INPUT_CONTROL.usa_TN_INPUT_CONTROL_DATA[1].by_Attr_oF := BYTE#16#74; (* Weiss, Blau *)
	Xus_TN_INPUT_CONTROL.usa_TN_INPUT_CONTROL_DATA[1].in_Cursor_Pos := INT#0;
	Xus_TN_INPUT_CONTROL.usa_TN_INPUT_CONTROL_DATA[1].bo_Input_Only_Num := FALSE;
	Xus_TN_INPUT_CONTROL.usa_TN_INPUT_CONTROL_DATA[1].bo_Input_Hidden := FALSE;
	Xus_TN_INPUT_CONTROL.usa_TN_INPUT_CONTROL_DATA[1].st_Input_Mask := '                                                                    ';
	Xus_TN_INPUT_CONTROL.usa_TN_INPUT_CONTROL_DATA[1].st_Input_Data := Xus_TN_INPUT_CONTROL.usa_TN_INPUT_CONTROL_DATA[1].st_Input_Mask;
	Xus_TN_INPUT_CONTROL.usa_TN_INPUT_CONTROL_DATA[1].st_Input_ToolTip := 'Eingabezeile aktiv       | SCROLL F1/F2/F3/F4 |';
	Xus_TN_INPUT_CONTROL.usa_TN_INPUT_CONTROL_DATA[1].in_Input_Option := INT#02;
	Xus_TN_INPUT_CONTROL.usa_TN_INPUT_CONTROL_DATA[1].in_Title_Y_Offset := INT#00;
	Xus_TN_INPUT_CONTROL.usa_TN_INPUT_CONTROL_DATA[1].in_Title_X_Offset := INT#00;
	Xus_TN_INPUT_CONTROL.usa_TN_INPUT_CONTROL_DATA[1].by_Title_Attr := BYTE#16#34;
	Xus_TN_INPUT_CONTROL.usa_TN_INPUT_CONTROL_DATA[1].st_Title_String := 'Befehl: ';

	(* Initialisierung Selection Text *)
	Xus_TN_INPUT_CONTROL.usa_TN_INPUT_CONTROL_DATA[2].in_Type := INT#03;
	Xus_TN_INPUT_CONTROL.usa_TN_INPUT_CONTROL_DATA[2].in_Y := INT#20;
	Xus_TN_INPUT_CONTROL.usa_TN_INPUT_CONTROL_DATA[2].in_X := INT#18;
	Xus_TN_INPUT_CONTROL.usa_TN_INPUT_CONTROL_DATA[2].by_Attr_mF := BYTE#16#17;
	Xus_TN_INPUT_CONTROL.usa_TN_INPUT_CONTROL_DATA[2].by_Attr_oF := BYTE#16#47;
	Xus_TN_INPUT_CONTROL.usa_TN_INPUT_CONTROL_DATA[2].st_Input_ToolTip := ' aktuellen LOG-Level aendern     | press enter to select |';
	Xus_TN_INPUT_CONTROL.usa_TN_INPUT_CONTROL_DATA[2].in_Input_Option := INT#00;
	Xus_TN_INPUT_CONTROL.usa_TN_INPUT_CONTROL_DATA[2].in_Title_Y_Offset := INT#00;
	Xus_TN_INPUT_CONTROL.usa_TN_INPUT_CONTROL_DATA[2].in_Title_X_Offset := INT#00;
	Xus_TN_INPUT_CONTROL.usa_TN_INPUT_CONTROL_DATA[2].by_Title_Attr := BYTE#16#34;
	Xus_TN_INPUT_CONTROL.usa_TN_INPUT_CONTROL_DATA[2].st_Title_String := ' LOG-Level ';
	Xus_TN_INPUT_CONTROL.usa_TN_INPUT_CONTROL_DATA[2].st_Input_Mask := '  ';
	Xus_TN_INPUT_CONTROL.usa_TN_INPUT_CONTROL_DATA[2].st_Input_Data := '01#02#03#04#05#06#07#08#09#10#11#12#13#14#15';

	(* Initialisierung Selection Text *)
	Xus_TN_INPUT_CONTROL.usa_TN_INPUT_CONTROL_DATA[3].in_Type := INT#02;
	Xus_TN_INPUT_CONTROL.usa_TN_INPUT_CONTROL_DATA[3].in_Y := INT#20;
	Xus_TN_INPUT_CONTROL.usa_TN_INPUT_CONTROL_DATA[3].in_X := INT#37;
	Xus_TN_INPUT_CONTROL.usa_TN_INPUT_CONTROL_DATA[3].by_Attr_mF := BYTE#16#17;
	Xus_TN_INPUT_CONTROL.usa_TN_INPUT_CONTROL_DATA[3].by_Attr_oF := BYTE#16#47;
	Xus_TN_INPUT_CONTROL.usa_TN_INPUT_CONTROL_DATA[3].st_Input_ToolTip := ' Optionline aktiv      | press space to select |';
	Xus_TN_INPUT_CONTROL.usa_TN_INPUT_CONTROL_DATA[3].in_Input_Option := INT#02;
	Xus_TN_INPUT_CONTROL.usa_TN_INPUT_CONTROL_DATA[3].in_Title_Y_Offset := INT#00;
	Xus_TN_INPUT_CONTROL.usa_TN_INPUT_CONTROL_DATA[3].in_Title_X_Offset := INT#00;
	Xus_TN_INPUT_CONTROL.usa_TN_INPUT_CONTROL_DATA[3].by_Title_Attr := BYTE#16#34;
	Xus_TN_INPUT_CONTROL.usa_TN_INPUT_CONTROL_DATA[3].st_Title_String := '  Selektion  ';
	Xus_TN_INPUT_CONTROL.usa_TN_INPUT_CONTROL_DATA[3].st_Input_Mask := '     ';
	Xus_TN_INPUT_CONTROL.usa_TN_INPUT_CONTROL_DATA[3].st_Input_Data := '[ ]#[x]';

	(* Initialisierung Selection Text *)
	Xus_TN_INPUT_CONTROL.usa_TN_INPUT_CONTROL_DATA[4].in_Type := INT#02;
	Xus_TN_INPUT_CONTROL.usa_TN_INPUT_CONTROL_DATA[4].in_Y := INT#20;
	Xus_TN_INPUT_CONTROL.usa_TN_INPUT_CONTROL_DATA[4].in_X := INT#58;
	Xus_TN_INPUT_CONTROL.usa_TN_INPUT_CONTROL_DATA[4].by_Attr_mF := BYTE#16#17;
	Xus_TN_INPUT_CONTROL.usa_TN_INPUT_CONTROL_DATA[4].by_Attr_oF := BYTE#16#47;
	Xus_TN_INPUT_CONTROL.usa_TN_INPUT_CONTROL_DATA[4].st_Input_ToolTip := ' Selektion-Text aktiv      | press space to select |';
	Xus_TN_INPUT_CONTROL.usa_TN_INPUT_CONTROL_DATA[4].in_Input_Option := INT#02;
	Xus_TN_INPUT_CONTROL.usa_TN_INPUT_CONTROL_DATA[4].in_Title_Y_Offset := INT#00;
	Xus_TN_INPUT_CONTROL.usa_TN_INPUT_CONTROL_DATA[4].in_Title_X_Offset := INT#00;
	Xus_TN_INPUT_CONTROL.usa_TN_INPUT_CONTROL_DATA[4].by_Title_Attr := BYTE#16#34;
	Xus_TN_INPUT_CONTROL.usa_TN_INPUT_CONTROL_DATA[4].st_Title_String := ' Betriebsart ';
	Xus_TN_INPUT_CONTROL.usa_TN_INPUT_CONTROL_DATA[4].st_Input_Mask := '               ';
	Xus_TN_INPUT_CONTROL.usa_TN_INPUT_CONTROL_DATA[4].st_Input_Data := '<Auto>#<Hand>#<Einzelschritt>#<Stop>#<Restart>';

	(* Control-Tool-Tip *)
	Xus_TN_INPUT_CONTROL.in_ToolTip_Y := INT#23;
	Xus_TN_INPUT_CONTROL.in_ToolTip_X := INT#00;
	Xus_TN_INPUT_CONTROL.by_ToolTip_Attr := BYTE#16#37;
	Xus_TN_INPUT_CONTROL.in_ToolTip_Size := INT#60;

	(* Control-Verwaltung initialisieren *)
	Xus_TN_INPUT_CONTROL.in_Count := INT#04;
	Xus_TN_INPUT_CONTROL.bo_Enable := TRUE;
	Xus_TN_INPUT_CONTROL.bo_Reset_Fokus := TRUE;

	(* LOG-Viewport initialisieren und Neuzeichnen auslösen *)
	us_LOG_VIEWPORT.COUNT := 13;
	us_LOG_VIEWPORT.UPDATE := TRUE;

	(* Menu initialisieren *)
	Xus_TN_MENU.in_X := INT#00;
	Xus_TN_MENU.in_Y := INT#00;
	Xus_TN_MENU.by_Attr_mF := BYTE#16#33; (* yellow + brown *)
	Xus_TN_MENU.by_Attr_oF := BYTE#16#0F; (* schwarz + grau *)
	Xus_TN_MENU.st_MENU_TEXT := 'Datei#Bearbeiten#Ansicht#Ende';
	Xus_TN_MENU.st_MENU_TEXT := CONCAT(Xus_TN_MENU.st_MENU_TEXT,'%oeffnen#-#speichern#beenden%loeschen#-#einfuegen#-#kopieren');
	Xus_TN_MENU.st_MENU_TEXT := CONCAT(Xus_TN_MENU.st_MENU_TEXT,'%alles#detail#kopieren%Logout');
	Xus_TN_MENU.bo_Create := TRUE;

END_IF;

IF (Xus_TN_SCREEN.in_Page_Number = INT#11) THEN

	(* Eingabezeile: Befehl -> eingegebenen String übernehmen *)
	IF (Xus_TN_INPUT_CONTROL.usa_TN_INPUT_CONTROL_DATA[1].bo_Input_Entered = TRUE) THEN

		Xus_TN_INPUT_CONTROL.usa_TN_INPUT_CONTROL_DATA[1].bo_Input_Entered := FALSE;
		Gst_SysLog_Command := Xus_TN_INPUT_CONTROL.usa_TN_INPUT_CONTROL_DATA[1].st_Input_String;

	END_IF;

	(* Eingabezeile: LOG_LEVEL -> eingegebenen String übernehmen *)
	IF (Xus_TN_INPUT_CONTROL.usa_TN_INPUT_CONTROL_DATA[2].bo_Input_Entered = TRUE) THEN

		Xus_TN_INPUT_CONTROL.usa_TN_INPUT_CONTROL_DATA[2].bo_Input_Entered := FALSE;
		Gst_SysLog_Command := CONCAT('LOG_LEVEL ',Xus_TN_INPUT_CONTROL.usa_TN_INPUT_CONTROL_DATA[2].st_Input_String);

	END_IF;

	(* LOG-Viewport - Scroll Funktionen *)
	IF (Xus_TN_INPUT_CONTROL.in_Focus_at = INT#01) THEN
		CASE BYTE_TO_INT(Xus_TN_SCREEN.by_Input_Exten_Code) OF
		80: (* F1 Taste *)
			us_LOG_VIEWPORT.MOVE_TO_X := 30001; (* Scrollen zum Listenanfang *)
		81: (* F2 Taste *)
			us_LOG_VIEWPORT.MOVE_TO_X := us_LOG_VIEWPORT.COUNT; (* Scrollen eine Seite nach oben *)
		82: (* F3 Taste *)
			us_LOG_VIEWPORT.MOVE_TO_X := 0 - us_LOG_VIEWPORT.COUNT;
		83: (* F4 Taste *)
			us_LOG_VIEWPORT.MOVE_TO_X := 30000; (* Scrollen zum Listenende *)
		END_CASE;
	END_IF;

	(* LOG-Viewport Updaten *)
	FB_LOG_VIEWPORT(LC := LOG_CL,
					LV := us_LOG_VIEWPORT);

	(* LOG-Viewport zeichnen *)
	FB_TN_SC_VIEWPORT(	Xus_LOG_VIEWPORT := us_LOG_VIEWPORT,
						Xus_LOG_CONTROL := LOG_CL,
						Xus_TN_SCREEN := Xus_TN_SCREEN,
						Iin_X := INT#01,
						Iin_Y := INT#02,
						Iin_Width := INT#76,
						Idw_ATTR_1 := DWORD#16#64542434, (* Color + Level 3:2:1:0 *)
						Idw_ATTR_2 := DWORD#16#94047414, (* Color + Level 7:6:5:4 *)
						Iti_TIME := TIME#100ms);
END_IF;

IF LEN(Gst_SysLog_Command) > 0 THEN

	(* Kommando echo *)
	LOG_CL.NEW_MSG := CONCAT('ACTION: ',Gst_SysLog_Command);
	LOG_CL.NEW_MSG_OPTION := 0;
	FB_LOG_MESSAGE();

	Gst_SysLog_Command := '';

END_IF;
END_PROGRAM

(* POU TN_FRAMEWORK, ST *)
FUNCTION_BLOCK TN_FRAMEWORK
VAR
	FB_IP_CONTROL : IP_CONTROL;
	FB_TN_INPUT_CONTROL : TN_INPUT_CONTROL;
	FB_TN_INPUT_MENU_BAR : TN_INPUT_MENU_BAR;
	FB_TN_RECEIVE :	TN_RECEIVE;
	FB_TN_SEND_ROWS : TN_SEND_ROWS;
	t : TON;
END_VAR
VAR_IN_OUT
	us_TN_INPUT_CONTROL : us_TN_INPUT_CONTROL;
	us_TN_SCREEN : us_TN_SCREEN;
	us_TN_MENU : us_TN_MENU;
	S_BUF : NETWORK_BUFFER;
	R_BUF : NETWORK_BUFFER;
	IP_C : IP_C;
END_VAR
VAR_INPUT
	PORT : WORD;
END_VAR

(*
version 1.1		17. may 2011
programmer		ks
tested by			ks

TN_FRAMEWORK ist ein Grundgerüst zur Nutzung des TELNET VISION Systems, und beinhält alle Laufzeit Komponenten.
*)
(* Initialisierung / Freigeben der Verbindung *)
IF (NOT IP_C.C_ENABLE) THEN

	(* IP Datenverkehr einrichten *)
	IP_C.C_PORT := SEL(PORT=BYTE#0,PORT,WORD#23); (* Portnummer eintragen *)
	IP_C.C_IP := DWORD#00; (* IP eintragen *)
	IP_C.C_MODE := BYTE#4; (* Mode: TCP+PASSIV+PORT *)
	IP_C.TIME_RESET := TRUE; (* Zeitueberwachung rücksetzen *)
	IP_C.C_ENABLE := TRUE; (* Verbindungsaufbau freigeben *)
	IP_C.R_OBSERVE := FALSE; (* keine Empfangsueberwachung *)

END_IF;

t(IN:= IP_C.ERROR > DWORD#0, PT:=T#5s);
IF t.Q THEN
	IP_C.TIME_RESET := TRUE; (* Error Reset *)
END_IF;

(* Telnet-Menu-Bar *)
FB_TN_INPUT_MENU_BAR(
	Xus_TN_MENU := us_TN_MENU,
	Xus_TN_SCREEN := us_TN_SCREEN);

(* Telnet-Input-Control *)
FB_TN_INPUT_CONTROL(
	Xus_TN_SCREEN := us_TN_SCREEN,
	Xus_TN_INPUT_CONTROL := us_TN_INPUT_CONTROL);

(* Telnet-Data-Send Line-Updates *)
FB_TN_SEND_ROWS(
	IP_C :=IP_C,
	S_BUF :=S_BUF,
	Xus_TN_SCREEN :=us_TN_SCREEN,
	S_BUF_SIZE :=SIZEOF(S_BUF.BUFFER));

(* Telnet-Server *)
FB_IP_CONTROL(
	IP_C :=IP_C,
	S_BUF :=S_BUF,
	R_BUF :=R_BUF,
	IP :=DWORD#00,
	PORT :=WORD#00,
	TIME_OUT :=T#2s);

(* Telnet-Data-Receive *)
FB_TN_RECEIVE(
	R_BUF := R_BUF,
	Xus_TN_SCREEN := us_TN_SCREEN);

(* revision history
ks	10. mai. 2010	rev 1.0
	original version

ks	17. may. 2011	rev 1.1
	automatischer re-connect

ks	05. may. 2012	rev 1.2
	neue parameter PORT
*)
END_FUNCTION_BLOCK

(* POU TN_INPUT_CONTROL, ST *)
FUNCTION_BLOCK TN_INPUT_CONTROL
VAR_IN_OUT
	Xus_TN_SCREEN : us_TN_SCREEN;
	Xus_TN_INPUT_CONTROL : us_TN_INPUT_CONTROL;
END_VAR
VAR
	FB_TN_INPUT_SELECT_POPUP : TN_INPUT_SELECT_POPUP;
	FB_TN_INPUT_SELECT_TEXT : TN_INPUT_SELECT_TEXT;
	FB_TN_SC_WRITE_C : TN_SC_WRITE_C;
	FB_TN_INPUT_EDIT_LINE : TN_INPUT_EDIT_LINE;
END_VAR
VAR
	in_index : INT;
	in_Scroll_Offset : INT;
	in_Focus_new : INT;
	in_Focus_alt : INT;
	bo_Tool_Tip_Update : BOOL;
END_VAR

(*
version 1.0		10. mai 2010
programmer		ks
tested by		ks

TN_INPUT_CONTROL dient zur verwaltung und grafischen Darstellung der INPUT_CONTROL Elemente
*)
(* Bearbeitung freigegeben ? *)
IF (Xus_TN_INPUT_CONTROL.bo_Enable = FALSE) OR (Xus_TN_SCREEN.bo_Menue_Bar_Dialog = TRUE) THEN
	RETURN;
END_IF;

(* Fokus Reset durchführen *)
IF (Xus_TN_INPUT_CONTROL.bo_Reset_Fokus = TRUE) THEN
	Xus_TN_INPUT_CONTROL.bo_Reset_Fokus := FALSE;

	FOR in_index := INT#01 TO Xus_TN_INPUT_CONTROL.in_Count DO
		Xus_TN_INPUT_CONTROL.usa_TN_INPUT_CONTROL_DATA[in_index].bo_Focus := FALSE;
	END_FOR;

	IF (Xus_TN_INPUT_CONTROL.in_Count >= INT#01) THEN
		Xus_TN_INPUT_CONTROL.usa_TN_INPUT_CONTROL_DATA[1].bo_Focus := TRUE;
		Xus_TN_INPUT_CONTROL.in_Focus_at := INT#01;
	END_IF;

	Xus_TN_INPUT_CONTROL.bo_Update_all := TRUE;
END_IF;

IF (Xus_TN_SCREEN.bo_Modal_Dialog = FALSE) THEN
	(* TAB-Taste für Control-element wechsel auswerten *)
	IF (Xus_TN_SCREEN.by_Input_Exten_Code = BYTE#09) THEN

		in_Scroll_Offset := INT#01;

		(* Cursor-Oben Taste *)
	ELSIF (Xus_TN_SCREEN.by_Input_Exten_Code = BYTE#65) THEN

		in_Scroll_Offset := -1;

		(* Cursor-unten Taste *)
	ELSIF (Xus_TN_SCREEN.by_Input_Exten_Code = BYTE#66) THEN

		in_Scroll_Offset := INT#01;

	END_IF;
END_IF;

IF (in_Scroll_Offset <> INT#00) THEN  
	(* Grenzwerte überprüfen                                            *)

	Xus_TN_INPUT_CONTROL.in_Focus_at:=LIMIT(INT#01,Xus_TN_INPUT_CONTROL.in_Focus_at,Xus_TN_INPUT_CONTROL.in_Count);

	in_Focus_new := Xus_TN_INPUT_CONTROL.in_Focus_at + in_Scroll_Offset;

	IF (in_Focus_new > Xus_TN_INPUT_CONTROL.in_Count) THEN
		in_Focus_new := INT#1;
	END_IF;

	IF (in_Focus_new < INT#01) THEN
		in_Focus_new := Xus_TN_INPUT_CONTROL.in_Count;
	END_IF;

	in_Focus_alt := Xus_TN_INPUT_CONTROL.in_Focus_at;

	(* aktuellen Element den Fokus entziehen *)
	Xus_TN_INPUT_CONTROL.usa_TN_INPUT_CONTROL_DATA[in_Focus_alt].bo_Focus := FALSE;
	Xus_TN_INPUT_CONTROL.usa_TN_INPUT_CONTROL_DATA[in_Focus_alt].bo_Update_Input := TRUE;

	(* neuem Element den Fokus geben *)
	Xus_TN_INPUT_CONTROL.usa_TN_INPUT_CONTROL_DATA[in_Focus_new].bo_Focus  := TRUE;
	Xus_TN_INPUT_CONTROL.usa_TN_INPUT_CONTROL_DATA[in_Focus_new].bo_Update_Input := TRUE;

	Xus_TN_INPUT_CONTROL.in_Focus_at := in_Focus_new;

	bo_Tool_Tip_Update := TRUE;
	in_Scroll_Offset := INT#00;

END_IF;

(* Alle Elemente updaten ? *)
IF (Xus_TN_INPUT_CONTROL.bo_Update_all = TRUE) THEN
	FOR in_index := 1 TO Xus_TN_INPUT_CONTROL.in_Count DO
		Xus_TN_INPUT_CONTROL.usa_TN_INPUT_CONTROL_DATA[in_index].bo_Update_All := TRUE;
	END_FOR;
	Xus_TN_INPUT_CONTROL.bo_Update_all := FALSE;
	bo_Tool_Tip_Update := TRUE;
END_IF;

FOR in_index := 1 TO Xus_TN_INPUT_CONTROL.in_Count DO

	IF (Xus_TN_INPUT_CONTROL.usa_TN_INPUT_CONTROL_DATA[in_index].in_Type > INT#00) THEN

		IF (Xus_TN_INPUT_CONTROL.usa_TN_INPUT_CONTROL_DATA[in_index].bo_Focus = TRUE) THEN

			Xus_TN_INPUT_CONTROL.usa_TN_INPUT_CONTROL_DATA[in_index].by_Input_ASCII_Code  := Xus_TN_SCREEN.by_Input_ASCII_Code;
			Xus_TN_INPUT_CONTROL.usa_TN_INPUT_CONTROL_DATA[in_index].by_Input_Exten_Code  := Xus_TN_SCREEN.by_Input_Exten_Code;
			Xus_TN_INPUT_CONTROL.usa_TN_INPUT_CONTROL_DATA[in_index].bo_Input_ASCII_IsNum := Xus_TN_SCREEN.bo_Input_ASCII_IsNum;

			(* Tool-Tip Text ausgeben *)
			IF (bo_Tool_Tip_Update = TRUE) THEN

				FB_TN_SC_WRITE_C(	Iin_Y := Xus_TN_INPUT_CONTROL.in_ToolTip_Y,
									Iin_X := Xus_TN_INPUT_CONTROL.in_ToolTip_X,
									Iby_ATTR := Xus_TN_INPUT_CONTROL.by_ToolTip_Attr,
									Iin_OPTION := INT#02, (* Center-String *)
									Iin_LENGTH := Xus_TN_INPUT_CONTROL.in_ToolTip_Size,
									Ist_STRING := Xus_TN_INPUT_CONTROL.usa_TN_INPUT_CONTROL_DATA[in_index].st_Input_ToolTip,
									Xus_TN_SCREEN := Xus_TN_SCREEN);

				(* Flag rücksetzen *)
				bo_Tool_Tip_Update := FALSE;
			END_IF;
		END_IF;

		CASE Xus_TN_INPUT_CONTROL.usa_TN_INPUT_CONTROL_DATA[in_index].in_Type OF
		1:
			(* Edit-Line bearbeiten *)
			FB_TN_INPUT_EDIT_LINE(	Xus_TN_INPUT_CONTROL_DATA := Xus_TN_INPUT_CONTROL.usa_TN_INPUT_CONTROL_DATA[in_index],
									Xus_TN_SCREEN := Xus_TN_SCREEN);
		2:
			(* Select-Text bearbeiten *)
			FB_TN_INPUT_SELECT_TEXT(	Xus_TN_INPUT_CONTROL_DATA := Xus_TN_INPUT_CONTROL.usa_TN_INPUT_CONTROL_DATA[in_index],
										Xus_TN_SCREEN := Xus_TN_SCREEN);
		3:
			(* Select-Popup bearbeiten *)
			FB_TN_INPUT_SELECT_POPUP(	Xus_TN_INPUT_CONTROL_DATA := Xus_TN_INPUT_CONTROL.usa_TN_INPUT_CONTROL_DATA[in_index],
										Xus_TN_SCREEN := Xus_TN_SCREEN);
		END_CASE;

		IF (Xus_TN_INPUT_CONTROL.usa_TN_INPUT_CONTROL_DATA[in_index].bo_Focus = TRUE) THEN

			(* Cursor position von Element auf Screen übertragen *)
			Xus_TN_SCREEN.in_Cursor_X := Xus_TN_INPUT_CONTROL.usa_TN_INPUT_CONTROL_DATA[in_index].in_Cursor_X;
			Xus_TN_SCREEN.in_Cursor_Y := Xus_TN_INPUT_CONTROL.usa_TN_INPUT_CONTROL_DATA[in_index].in_Cursor_Y;

		END_IF;
	END_IF;
END_FOR;

(* revision history
ks	10. mai. 2010	rev 1.0
	original version
*)
END_FUNCTION_BLOCK

(* POU TN_INPUT_SELECT_POPUP, ST *)
FUNCTION_BLOCK TN_INPUT_SELECT_POPUP
VAR
	in_index : INT;
	in_Element_Count : INT;
	by_Cur_Key : BYTE;
	by_Attr : BYTE;
	st_String : STRING;
END_VAR
VAR
	us_TN_MENU_POPUP : us_TN_MENU_POPUP;
	FB_TN_INPUT_MENU_POPUP : TN_INPUT_MENU_POPUP;
	FB_TN_SC_WRITE : TN_SC_WRITE;
END_VAR
VAR_IN_OUT
	Xus_TN_SCREEN : us_TN_SCREEN;
	Xus_TN_INPUT_CONTROL_DATA : us_TN_INPUT_CONTROL_DATA;
END_VAR

(*
version 1.1		06. apr 2011
programmer		ks
tested by			ks

TN_SELECT_POPUP dient zur verwaltung und darstellung eines POPUP-Dialogs zur Elementeauswahl
*)
(* Benutzereingabe auswerten -> Selektion Text n *)
IF (Xus_TN_INPUT_CONTROL_DATA.bo_Focus = TRUE) THEN

	by_Cur_Key := Xus_TN_INPUT_CONTROL_DATA.by_Input_Exten_Code;

	IF (us_TN_MENU_POPUP.bo_Activ = FALSE) THEN
		us_TN_MENU_POPUP.by_Input_Exten_Code := BYTE#00;

		(* Return-Taste auswerten *)
		IF (by_Cur_Key = BYTE#13) THEN
			(* Popup-Menu parameter übergeben *)
			us_TN_MENU_POPUP.in_Y := Xus_TN_INPUT_CONTROL_DATA.in_Y;
			us_TN_MENU_POPUP.in_X := Xus_TN_INPUT_CONTROL_DATA.in_X;
			us_TN_MENU_POPUP.by_Attr_mF := Xus_TN_INPUT_CONTROL_DATA.by_Attr_mF;
			us_TN_MENU_POPUP.by_Attr_oF := Xus_TN_INPUT_CONTROL_DATA.by_Attr_oF;
			us_TN_MENU_POPUP.st_Menu_Text := Xus_TN_INPUT_CONTROL_DATA.st_Input_Data;
			us_TN_MENU_POPUP.bo_Create := TRUE;
			us_TN_MENU_POPUP.in_Cur_Item := INT#00;
		END_IF;

		IF (us_TN_MENU_POPUP.in_Cur_Item > INT#00) THEN
			Xus_TN_INPUT_CONTROL_DATA.in_selected := us_TN_MENU_POPUP.in_Cur_Item;
			Xus_TN_INPUT_CONTROL_DATA.bo_Input_Entered := TRUE;
			Xus_TN_INPUT_CONTROL_DATA.bo_Update_Input := TRUE;
			us_TN_MENU_POPUP.in_Cur_Item := INT#00;
		END_IF;

	ELSE
		us_TN_MENU_POPUP.by_Input_Exten_Code := by_Cur_Key;
	END_IF;

	(* Popup-Menu zyklisch aufrufen *)
	FB_TN_INPUT_MENU_POPUP(Xus_TN_MENU_POPUP := us_TN_MENU_POPUP, Xus_TN_SCREEN := Xus_TN_SCREEN);

END_IF;

(* Aktualisierung der Anzeige *)
IF (Xus_TN_INPUT_CONTROL_DATA.bo_Update_Input = TRUE) OR (Xus_TN_INPUT_CONTROL_DATA.bo_Update_All = TRUE) THEN

	(* Title-Text ausgeben *)
	IF Xus_TN_INPUT_CONTROL_DATA.bo_Update_All = TRUE THEN

		IF (Xus_TN_INPUT_CONTROL_DATA.in_Title_X_Offset = INT#00) AND (Xus_TN_INPUT_CONTROL_DATA.in_Title_Y_Offset = INT#00) THEN
			(* wenn Offset X,Y =0 dann Titlestring links vom Element positionieren *)
			FB_TN_SC_WRITE.Iin_Y := Xus_TN_INPUT_CONTROL_DATA.in_Y;
			FB_TN_SC_WRITE.Iin_X := Xus_TN_INPUT_CONTROL_DATA.in_X - LEN(Xus_TN_INPUT_CONTROL_DATA.st_Title_String);

		ELSE
			(* Title-Text durch Row, Color-Offset ausgeben *)
			FB_TN_SC_WRITE.Iin_Y := Xus_TN_INPUT_CONTROL_DATA.in_Y + Xus_TN_INPUT_CONTROL_DATA.in_Title_Y_Offset;
			FB_TN_SC_WRITE.Iin_X := Xus_TN_INPUT_CONTROL_DATA.in_X + Xus_TN_INPUT_CONTROL_DATA.in_Title_X_Offset;
		END_IF;

		(* Title-Text durch Row, Color-Offset ausgeben *)
		FB_TN_SC_WRITE(	Iby_ATTR := Xus_TN_INPUT_CONTROL_DATA.by_Title_Attr,
						Ist_STRING := Xus_TN_INPUT_CONTROL_DATA.st_Title_String,
						Xus_TN_SCREEN := Xus_TN_SCREEN);
	END_IF;

	in_Element_Count := ELEMENT_COUNT(SEP:=BYTE#35,ELEMENT:=Xus_TN_INPUT_CONTROL_DATA.st_Input_Data);

	IF in_Element_Count > INT#00 THEN

		Xus_TN_INPUT_CONTROL_DATA.in_selected:=LIMIT(1,Xus_TN_INPUT_CONTROL_DATA.in_selected,in_Element_Count);

		in_index := Xus_TN_INPUT_CONTROL_DATA.in_selected;

		st_String := ELEMENT_GET(SEP:=BYTE#35,POS:=in_index - 1,ELEMENT:=Xus_TN_INPUT_CONTROL_DATA.st_Input_Data);

		st_String:= FIX(str:=st_String,
						L:=LEN(Xus_TN_INPUT_CONTROL_DATA.st_Input_Mask),
						C:=BYTE#32,
						M:=Xus_TN_INPUT_CONTROL_DATA.in_Input_Option);


		Xus_TN_INPUT_CONTROL_DATA.st_Input_String := st_String;

		IF Xus_TN_INPUT_CONTROL_DATA.bo_Focus = TRUE THEN
			by_Attr := Xus_TN_INPUT_CONTROL_DATA.by_Attr_mF;
		ELSE
			by_Attr := Xus_TN_INPUT_CONTROL_DATA.by_Attr_oF;
		END_IF;

		FB_TN_SC_WRITE(	Iin_X := Xus_TN_INPUT_CONTROL_DATA.in_X,
								Iin_Y := Xus_TN_INPUT_CONTROL_DATA.in_Y,
								Iby_ATTR := by_Attr,
								Ist_STRING := st_String,
								Xus_TN_SCREEN := Xus_TN_SCREEN );
	END_IF;

	(* Cursor auf aktuelle Position setzen *)
	Xus_TN_INPUT_CONTROL_DATA.in_Cursor_X := Xus_TN_INPUT_CONTROL_DATA.in_X;
	Xus_TN_INPUT_CONTROL_DATA.in_Cursor_Y := Xus_TN_INPUT_CONTROL_DATA.in_Y;

	(* Update-Flag's rücksetzen *)
	Xus_TN_INPUT_CONTROL_DATA.bo_Update_All   := FALSE;
	Xus_TN_INPUT_CONTROL_DATA.bo_Update_Input := FALSE;

END_IF;

(* revision history

ks	06. apr. 2011	rev 1.1
	list_len und list_get durch element_count und element_get ersetzt

ks	10. mai. 2010	rev 1.0
	original version
*)
END_FUNCTION_BLOCK

(* POU TN_INPUT_MENU_POPUP, ST *)
FUNCTION_BLOCK TN_INPUT_MENU_POPUP
VAR
	FB_TN_SC_AREA_SAVE : TN_SC_AREA_SAVE;
	FB_TN_SC_AREA_RESTORE : TN_SC_AREA_RESTORE;
	FB_TN_SC_LINE : TN_SC_LINE;
	FB_TN_SC_ADD_SHADOW : TN_SC_ADD_SHADOW;
	FB_TN_SC_BOX : TN_SC_BOX;
	FB_TN_SC_WRITE_C : TN_SC_WRITE_C;
END_VAR
VAR
	in_ROW : INT;
	in_ROWS : INT;
	in_COL : INT;
	in_COLS : INT;
	in_index : INT;
	in_Count : INT;
	in_Scroll_Offset : INT;
	by_ATTR : BYTE;
END_VAR
VAR_IN_OUT
	Xus_TN_MENU_POPUP : us_TN_MENU_POPUP;
	Xus_TN_SCREEN : us_TN_SCREEN;
END_VAR

(*
version 1.1		06. apr 2011
programmer		ks
tested by			ks

TN_MENU_POPUP dient zur verwaltung und darstellung eines MENU-POPUP
*)
(* sicherstellen das rechteck immer innerhalb screen positioniert wird *)

IF (Xus_TN_MENU_POPUP.bo_Activ = FALSE) AND (Xus_TN_MENU_POPUP.bo_Create = TRUE) THEN
	Xus_TN_MENU_POPUP.bo_Activ := TRUE;
	Xus_TN_MENU_POPUP.bo_Create := FALSE;
	Xus_TN_MENU_POPUP.bo_Destroy := FALSE;
	Xus_TN_MENU_POPUP.bo_Update := TRUE;

  (* Sub-Menu-Texte *)

	Xus_TN_MENU_POPUP.in_Menu_E_Count := ELEMENT_COUNT(SEP:=BYTE#35,ELEMENT:=Xus_TN_MENU_POPUP.st_Menu_Text);

	(* Anzahl Zeilen (Sub-Menu-Texte) bestimmen *)
	Xus_TN_MENU_POPUP.in_Rows := Xus_TN_MENU_POPUP.in_Menu_E_Count;

	(* längsten Sub-Menu-Text suchen *)
	Xus_TN_MENU_POPUP.in_Cols := INT#00;

	FOR in_Count := INT#01 TO Xus_TN_MENU_POPUP.in_Rows DO;
		Xus_TN_MENU_POPUP.in_Cols:=MAX(LEN(ELEMENT_GET(SEP:=BYTE#35,POS:=in_Count - 1,ELEMENT:=Xus_TN_MENU_POPUP.st_Menu_Text)),Xus_TN_MENU_POPUP.in_Cols);
	END_FOR;

	(* Horizontale Position überprüfen und korrigieren *)
	IF (Xus_TN_MENU_POPUP.in_X + Xus_TN_MENU_POPUP.in_Cols) > INT#75 THEN
		Xus_TN_MENU_POPUP.in_X := INT#79 - Xus_TN_MENU_POPUP.in_Cols - INT#04;
	END_IF;

  (* Vertikale Position überprüfen und korrigieren *)
	IF (Xus_TN_MENU_POPUP.in_Y + Xus_TN_MENU_POPUP.in_ROWS) > INT#21 THEN
		Xus_TN_MENU_POPUP.in_Y := INT#23 - Xus_TN_MENU_POPUP.in_ROWS - INT#2;
	END_IF;

	Xus_TN_SCREEN.bo_Modal_Dialog := TRUE;

	(* Hintergrund sichern *)
	FB_TN_SC_AREA_SAVE(	Iin_X1 := Xus_TN_MENU_POPUP.in_X,
									Iin_Y1 := Xus_TN_MENU_POPUP.in_Y,
									Iin_X2 := Xus_TN_MENU_POPUP.in_X + Xus_TN_MENU_POPUP.in_Cols + INT#04,
									Iin_Y2 := Xus_TN_MENU_POPUP.in_Y + Xus_TN_MENU_POPUP.in_Rows + INT#02,
									Xus_TN_SCREEN := Xus_TN_SCREEN);

	(* Rahmen für Submenu zeichnen *)
	FB_TN_SC_BOX(	Iin_X1 := Xus_TN_MENU_POPUP.in_X,
					Iin_Y1 := Xus_TN_MENU_POPUP.in_Y,
					Iin_X2 := Xus_TN_MENU_POPUP.in_X + Xus_TN_MENU_POPUP.in_Cols + INT#03,
					Iin_Y2 := Xus_TN_MENU_POPUP.in_Y + Xus_TN_MENU_POPUP.in_Rows + INT#01,
					Iby_FILL := BYTE#32, (* Füllung *)
					Iin_BORDER := INT#01, (* Single-Line Border *)
					Iby_ATTR := Xus_TN_MENU_POPUP.by_Attr_oF,
					Xus_TN_SCREEN := Xus_TN_SCREEN);

	(* Shadow für Submenu zeichnen *)
	FB_TN_SC_ADD_SHADOW(Iin_X1 := Xus_TN_MENU_POPUP.in_X + INT#1,
						Iin_Y1 := Xus_TN_MENU_POPUP.in_Y + INT#1,
						Iin_X2 := Xus_TN_MENU_POPUP.in_X + Xus_TN_MENU_POPUP.in_Cols + INT#04,
						Iin_Y2 := Xus_TN_MENU_POPUP.in_Y + Xus_TN_MENU_POPUP.in_Rows + INT#02,
						Iin_OPTION := INT#00,
						Xus_TN_SCREEN := Xus_TN_SCREEN);

	(* Parameter laden *)
	in_COL := Xus_TN_MENU_POPUP.in_X;
	in_ROW := Xus_TN_MENU_POPUP.in_Y;
	in_ROWS := Xus_TN_MENU_POPUP.in_Rows;
	in_COLS := Xus_TN_MENU_POPUP.in_Cols;

	(* Trennlinien zeichnen *)
	in_COLS := in_COLS + INT#02; (* Text um 2 Zeichen verlängern *)

	FOR in_Count := INT#01 TO Xus_TN_MENU_POPUP.in_Menu_E_Count DO;
		in_ROW := in_ROW + INT#01;

		IF ELEMENT_GET(SEP:=BYTE#35,POS:=in_Count - 1,ELEMENT:=Xus_TN_MENU_POPUP.st_Menu_Text) = '-' THEN

			FB_TN_SC_LINE(	Iin_Y1 := in_ROW,
							Iin_X1 := in_COL,
							Iin_Y2 := in_ROW,
							Iin_X2 := in_COL + in_COLS + INT#01,
							Iby_ATTR := Xus_TN_MENU_POPUP.by_Attr_oF,
							Iby_BORDER := BYTE#01,
							Xus_TN_SCREEN := Xus_TN_SCREEN);
		END_IF;
	END_FOR;
END_IF;

IF (Xus_TN_MENU_POPUP.bo_Activ = TRUE) THEN

	CASE BYTE_TO_INT(Xus_TN_MENU_POPUP.by_Input_Exten_Code) OF

	65: (* Cursor oben *)
		in_Scroll_Offset := -1;
		Xus_TN_MENU_POPUP.bo_Update := TRUE;

	66: (* Cursor unten *)
		in_Scroll_Offset := 1;
		Xus_TN_MENU_POPUP.bo_Update := TRUE;

	13:  (* Enter *)
		Xus_TN_MENU_POPUP.bo_Destroy := TRUE;

	27:  (* Escape*)
		Xus_TN_MENU_POPUP.bo_Destroy := TRUE;
		Xus_TN_MENU_POPUP.in_Cur_Item := INT#00;

	67..68: (* Cursor links oder rechts *)
		Xus_TN_MENU_POPUP.bo_Destroy := TRUE;
		Xus_TN_MENU_POPUP.in_Cur_Item := INT#00;

	END_CASE;
END_IF;

(* POPUP-Menu updaten *)
IF (Xus_TN_MENU_POPUP.bo_Activ = TRUE) AND (Xus_TN_MENU_POPUP.bo_Update = TRUE) THEN

	Xus_TN_MENU_POPUP.bo_Update := FALSE;

	(* überprüfung + nächstes anwählbares Sub-Menu suchen *)
	in_index := Xus_TN_MENU_POPUP.in_Cur_Item;

	IF (in_index < INT#01) OR (in_index > Xus_TN_MENU_POPUP.in_Menu_E_Count) THEN
		in_Scroll_Offset := INT#01;
		in_index := Xus_TN_MENU_POPUP.in_Menu_E_Count;
	END_IF;

	(* aktueller Index steht auf Trennzeichen -> ändern *)
	IF ELEMENT_GET(SEP:=BYTE#35,POS:=in_index-1,ELEMENT:=Xus_TN_MENU_POPUP.st_Menu_Text) = '-' THEN
		in_Scroll_Offset := INT#01;
	END_IF;

	(* Scroll-Offset *)
	IF in_Scroll_Offset <> INT#00 THEN

		FOR in_Count := INT#01 TO Xus_TN_MENU_POPUP.in_Menu_E_Count DO;

			in_index:=INC2(in_index,in_Scroll_Offset,1,Xus_TN_MENU_POPUP.in_Menu_E_Count);

			IF ELEMENT_GET(SEP:=BYTE#35,POS:=in_index - 1,ELEMENT:=Xus_TN_MENU_POPUP.st_Menu_Text) <> '-' THEN
				EXIT;
			END_IF;

		END_FOR;
	END_IF;

	Xus_TN_MENU_POPUP.in_Cur_Item := in_index;
	in_Scroll_Offset := INT#00;

	(* Parameter laden *)
	in_COL  := Xus_TN_MENU_POPUP.in_X;
	in_ROW  := Xus_TN_MENU_POPUP.in_Y;
	in_ROWS := Xus_TN_MENU_POPUP.in_Rows;
	in_COLS := Xus_TN_MENU_POPUP.in_Cols;

	(* SUB-MENU-Titel ausgeben *)
	in_COLS := in_COLS + INT#02; (* Text um 2 Zeichen verlängern *)

	FOR in_Count := INT#01 TO Xus_TN_MENU_POPUP.in_Menu_E_Count DO;

		in_ROW := in_ROW + INT#01;

		(* Zeichenfarbe bestimmen *)
		IF in_Count = Xus_TN_MENU_POPUP.in_Cur_Item THEN
			by_ATTR := Xus_TN_MENU_POPUP.by_Attr_mF;
		ELSE
			by_ATTR := Xus_TN_MENU_POPUP.by_Attr_oF;
		END_IF;

		FB_TN_SC_WRITE_C.Ist_STRING := ELEMENT_GET(SEP:=BYTE#35,POS:=in_Count - 1,ELEMENT:=Xus_TN_MENU_POPUP.st_Menu_Text);

		IF FB_TN_SC_WRITE_C.Ist_STRING <> '-' THEN

			FB_TN_SC_WRITE_C(	Iin_Y := in_ROW,
								Iin_X := in_COL + INT#01,
								Iby_ATTR := by_ATTR,
								Iin_LENGTH := in_COLS,
								Iin_OPTION := INT#02, (* Center *)
								Xus_TN_SCREEN := Xus_TN_SCREEN);
		END_IF;
	END_FOR;
END_IF;

(* POPUP-Menu entfernen (Destroy) *)
IF (Xus_TN_MENU_POPUP.bo_Activ = TRUE) AND (Xus_TN_MENU_POPUP.bo_Destroy = TRUE) THEN

	Xus_TN_MENU_POPUP.bo_Destroy := FALSE;
	Xus_TN_MENU_POPUP.bo_Activ := FALSE;

	(* alten Hintergrund aus Speicher wiederherstellen *)
	FB_TN_SC_AREA_RESTORE(Xus_TN_SCREEN := Xus_TN_SCREEN);

	Xus_TN_SCREEN.bo_Modal_Dialog := FALSE;
END_IF;

(* revision history

ks	06. apr. 2011	rev 1.1
	list_len und list_get durch element_count und element_get ersetzt

ks	10. mai. 2010	rev 1.0
	original version
*)
END_FUNCTION_BLOCK

(* POU TN_SC_AREA_SAVE, ST *)
FUNCTION_BLOCK TN_SC_AREA_SAVE
VAR
	in_Offset_1 : INT;
	in_Offset_2 : INT;
	in_Y : INT;
	in_X : INT;
END_VAR
VAR_INPUT
	Iin_Y1 : INT;
	Iin_X1 : INT;
	Iin_Y2 : INT;
	Iin_X2 : INT;
END_VAR
VAR_IN_OUT
	Xus_TN_SCREEN : us_TN_SCREEN;
END_VAR

(*
version 1.0		10. mai 2010
programmer		ks
tested by		ks

TN_SC_AREA_SAVE sichert den angegebenen Bildschirmbereich in einem Buffer
*)
IF TN_SC_XY2_ERROR(Iin_X1,Iin_Y1,Iin_X2,Iin_Y2) THEN RETURN; END_IF;

(* Parameter ablegen *)
Xus_TN_SCREEN.bya_BACKUP[0] := BYTE#1;
Xus_TN_SCREEN.bya_BACKUP[1] := INT_TO_BYTE(Iin_X1);
Xus_TN_SCREEN.bya_BACKUP[2] := INT_TO_BYTE(Iin_Y1); 
Xus_TN_SCREEN.bya_BACKUP[3] := INT_TO_BYTE(Iin_X2);
Xus_TN_SCREEN.bya_BACKUP[4] := INT_TO_BYTE(Iin_Y2);

in_Offset_2 := 5;
(* CHAR und COLOR in BUFFER sichern *)
FOR in_Y := Iin_Y1 TO Iin_Y2 DO

	in_Offset_1 := (in_Y * 80) + Iin_X1;
	FOR in_X := Iin_X1 TO Iin_X2 DO
		Xus_TN_SCREEN.bya_BACKUP[in_Offset_2] := Xus_TN_SCREEN.bya_CHAR[in_Offset_1];
		in_Offset_2 := in_Offset_2 + INT#01;
		Xus_TN_SCREEN.bya_BACKUP[in_Offset_2] := Xus_TN_SCREEN.bya_COLOR[in_Offset_1];
		in_Offset_2 := in_Offset_2 + INT#01;
		in_Offset_1 := in_Offset_1 + INT#01;
	END_FOR;
END_FOR;

(* revision history
ks	10. mai. 2010	rev 1.0
	original version
*)
END_FUNCTION_BLOCK

(* POU TN_SC_XY2_ERROR, ST *)
FUNCTION TN_SC_XY2_ERROR : BOOL
VAR_INPUT
	X1 : INT;
	Y1 : INT;
	X2 : INT;
	Y2 : INT;
END_VAR

(*
version 1.0		10. mai 2010
programmer		ks
tested by		ks

TN_SC_XY2_ERROR prüft ob die angegenene Koordinaten die einen rechteckigen Bereich angeben gültig sind 
*)
(* min und max werte prüfen *)
TN_SC_XY2_ERROR := Y1 < 0 OR X1 < 0 OR Y2 < 0 OR X2 < 0 OR Y1 > 23 OR X1 > 79 OR Y2 > 23 OR X2 > 79;

(* revision history
ks	10. mai. 2010	rev 1.0
	original version
*)
END_FUNCTION

(* POU TN_SC_AREA_RESTORE, ST *)
FUNCTION_BLOCK TN_SC_AREA_RESTORE
VAR
	in_Offset_1 : INT;
	in_Offset_2 : INT;
	in_Y : INT;
	in_X : INT;
	in_Y1 : INT;
	in_X1 : INT;
	in_Y2 : INT;
	in_X2 : INT;
END_VAR
VAR_IN_OUT
	Xus_TN_SCREEN : us_TN_SCREEN;
END_VAR

(*
version 1.0		10. mai 2010
programmer		ks
tested by		ks

TN_SC_AREA_RESTORE stellt den zuvor gesicherten Bildschirmbereich wieder her
*)
IF Xus_TN_SCREEN.bya_BACKUP[0] > BYTE#00 THEN

	(* Parameter auslesen *)
	in_X1 := BYTE_TO_INT(Xus_TN_SCREEN.bya_BACKUP[1]);
	in_Y1 := BYTE_TO_INT(Xus_TN_SCREEN.bya_BACKUP[2]);
	in_X2 := BYTE_TO_INT(Xus_TN_SCREEN.bya_BACKUP[3]);
	in_Y2 := BYTE_TO_INT(Xus_TN_SCREEN.bya_BACKUP[4]);

	IF TN_SC_XY2_ERROR(in_X1,in_Y1,in_X2,in_Y2) THEN RETURN; END_IF;
	in_Offset_2 := 5;

	(* CHAR und COLOR von BUFFER wiederherstellen *)
	FOR in_Y := in_Y1 TO in_Y2 DO

		Xus_TN_SCREEN.bya_Line_Update[in_Y] := TRUE; (* Zeile zum Updaten freigeben *)
		in_Offset_1 := (in_Y * 80) + in_X1;

		FOR in_X := in_X1 TO in_X2 DO

			Xus_TN_SCREEN.bya_CHAR[in_Offset_1] := Xus_TN_SCREEN.bya_BACKUP[in_Offset_2];
			in_Offset_2 := in_Offset_2 + INT#01;

			Xus_TN_SCREEN.bya_COLOR[in_Offset_1] := Xus_TN_SCREEN.bya_BACKUP[in_Offset_2];
			in_Offset_2 := in_Offset_2 + INT#01;
			in_Offset_1 := in_Offset_1 + INT#01;

		END_FOR;
	END_FOR;

	(* Daten als ungültig markieren *)
	Xus_TN_SCREEN.bya_BACKUP[0] := BYTE#00;
END_IF;

(* revision history
ks	10. mai. 2010	rev 1.0
	original version
*)
END_FUNCTION_BLOCK

(* POU TN_SC_LINE, ST *)
FUNCTION_BLOCK TN_SC_LINE
VAR
	by_Connect_Left_Char : BYTE;
	by_Connect_Right_Char : BYTE;
	by_Connect_Top_Char : BYTE;
	by_Connect_Bottom_Char : BYTE;
	by_Connect_Cruz_Char : BYTE;
	by_Vertikal_Line_Char : BYTE;
	by_Horzontal_Line_Char : BYTE;
	by_old_Char : BYTE;
	in_Offset_1 : INT;
	in_ROW_Index : INT;
	in_COL_Index : INT;
	by_Char : BYTE;
END_VAR
VAR_INPUT
	Iin_X1 : INT;
	Iin_Y1 : INT;
	Iin_X2 : INT;
	Iin_Y2 : INT;
	Iby_ATTR : BYTE;
	Iby_BORDER : BYTE;
END_VAR
VAR_IN_OUT
	Xus_TN_SCREEN : us_TN_SCREEN;
END_VAR

(*
version 1.0		10. mai 2010
programmer		ks
tested by		ks

TN_SC_LINE zeichnet horizontale und vertikale Linien
*)
IF TN_SC_XY2_ERROR(Iin_X1,Iin_Y1,Iin_X2,Iin_Y2) THEN RETURN; END_IF;

(* Bordertype bestimmen *)
IF Iby_Border = BYTE#01 THEN (* Single Line *)
	by_Connect_Top_Char := BYTE#16#C2;
	by_Connect_Bottom_Char := BYTE#16#C1;
	by_Connect_Left_Char := BYTE#16#C3;
	by_Connect_Right_Char := BYTE#16#B4;
	by_Horzontal_Line_Char := BYTE#16#C4;
	by_Vertikal_Line_Char := BYTE#16#B3;
	by_Connect_Cruz_Char := BYTE#16#C5;
ELSIF Iby_Border = BYTE#02 THEN	(* Double Linie *)
	by_Connect_Top_Char := BYTE#16#CB;
	by_Connect_Bottom_Char := BYTE#16#CA;
	by_Connect_Left_Char := BYTE#16#CC;
	by_Connect_Right_Char := BYTE#16#B9;
	by_Horzontal_Line_Char := BYTE#16#CD;
	by_Vertikal_Line_Char := BYTE#16#BA;
	by_Connect_Cruz_Char := BYTE#16#CE;
ELSE (* Full Linie *)
	by_Connect_Top_Char := Iby_Border;
	by_Connect_Bottom_Char := Iby_Border;
	by_Connect_Left_Char := Iby_Border;
	by_Connect_Right_Char := Iby_Border;
	by_Horzontal_Line_Char := Iby_Border;
	by_Vertikal_Line_Char := Iby_Border;
	by_Connect_Cruz_Char := Iby_Border;
END_IF;

